ABB RAPID module: arm_code.mod

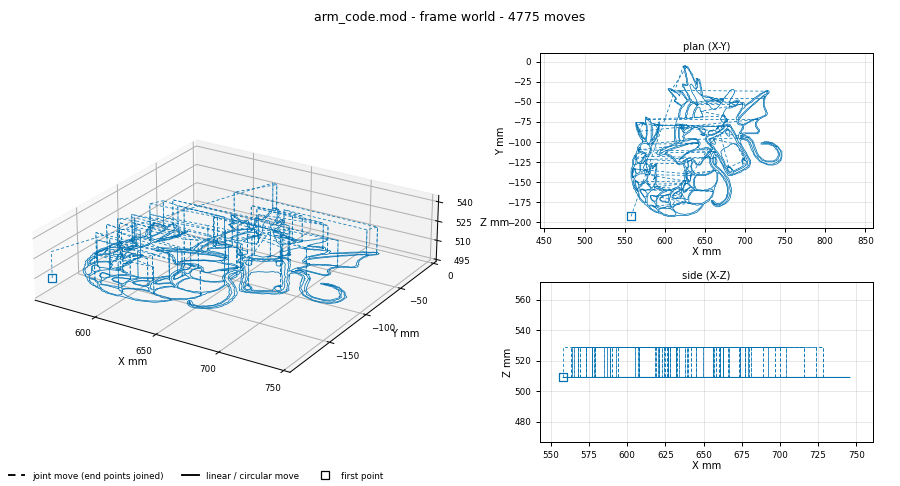
[picture p0: tool path of arm_code.mod in frame world, 4775 of 4775 moves have a stored position in this frame; points joined in program order, loops and branches not executed]
MODULE Module1
    !***********************************************************
    !
    ! Module:  Module1
    !
    ! Description:
    !   <Insert description here>
    !
    ! Author: ufabc
    !
    ! Version: 1.0
    !
    !***********************************************************


    !***********************************************************
    !
    ! Procedure main
    !
    !   This is the entry point of your program
    !
    !***********************************************************
    PROC main()
        !Add your code here
        CONST robtarget p0:=[[557.96,-192.62,509.20],[0.00299687,-0.165444,-0.986215,-0.000502744],[-1,0,0,0],[9E+09,9E+09,9E+09,9E+09,9E+09,9E+09]]
;
        MoveJ p0, v10, z1, tool0;
	MoveJ Offs(p0,0,0, 20), v10, z1, tool0;
	MoveJ Offs(p0,65.0,187.0, 20), v10, z1, tool0;
	MoveJ Offs(p0,65.0,187.0, 0), v10, z1, tool0;
	MoveL Offs(p0,66.0,184.0, 0), v10, z5, tool0;
	MoveL Offs(p0,66.0,184.0, 0), v10, z5, tool0;
	MoveL Offs(p0,66.0,184.0, 0), v10, z5, tool0;
	MoveL Offs(p0,67.0,181.0, 0), v10, z5, tool0;
	MoveL Offs(p0,67.0,179.0, 0), v10, z5, tool0;
	MoveL Offs(p0,68.0,176.0, 0), v10, z5, tool0;
	MoveL Offs(p0,68.0,174.0, 0), v10, z5, tool0;
	MoveL Offs(p0,69.0,172.0, 0), v10, z5, tool0;
	MoveL Offs(p0,69.0,169.0, 0), v10, z5, tool0;
	MoveL Offs(p0,69.0,167.0, 0), v10, z5, tool0;
	MoveL Offs(p0,70.0,165.0, 0), v10, z5, tool0;
	MoveL Offs(p0,70.0,164.0, 0), v10, z5, tool0;
	MoveL Offs(p0,70.0,163.0, 0), v10, z5, tool0;
	MoveL Offs(p0,68.0,164.0, 0), v10, z5, tool0;
	MoveL Offs(p0,66.0,165.0, 0), v10, z5, tool0;
	MoveL Offs(p0,65.0,165.0, 0), v10, z5, tool0;
	MoveL Offs(p0,65.0,165.0, 0), v10, z5, tool0;
	MoveL Offs(p0,64.0,165.0, 0), v10, z5, tool0;
	MoveL Offs(p0,64.0,165.0, 0), v10, z5, tool0;
	MoveL Offs(p0,64.0,165.0, 0), v10, z5, tool0;
	MoveL Offs(p0,64.0,165.0, 0), v10, z5, tool0;
	MoveL Offs(p0,64.0,162.0, 0), v10, z5, tool0;
	MoveL Offs(p0,65.0,161.0, 0), v10, z5, tool0;
	MoveL Offs(p0,65.0,161.0, 0), v10, z5, tool0;
	MoveL Offs(p0,66.0,160.0, 0), v10, z5, tool0;
	MoveL Offs(p0,68.0,156.0, 0), v10, z5, tool0;
	MoveL Offs(p0,69.0,155.0, 0), v10, z5, tool0;
	MoveL Offs(p0,70.0,153.0, 0), v10, z5, tool0;
	MoveL Offs(p0,70.0,151.0, 0), v10, z5, tool0;
	MoveL Offs(p0,71.0,150.0, 0), v10, z5, tool0;
	MoveL Offs(p0,72.0,149.0, 0), v10, z5, tool0;
	MoveL Offs(p0,72.0,147.0, 0), v10, z5, tool0;
	MoveL Offs(p0,73.0,147.0, 0), v10, z5, tool0;
	MoveL Offs(p0,73.0,146.0, 0), v10, z5, tool0;
	MoveL Offs(p0,71.0,145.0, 0), v10, z5, tool0;
	MoveL Offs(p0,69.0,147.0, 0), v10, z5, tool0;
	MoveL Offs(p0,69.0,148.0, 0), v10, z5, tool0;
	MoveL Offs(p0,68.0,148.0, 0), v10, z5, tool0;
	MoveL Offs(p0,67.0,151.0, 0), v10, z5, tool0;
	MoveL Offs(p0,66.0,152.0, 0), v10, z5, tool0;
	MoveL Offs(p0,66.0,152.0, 0), v10, z5, tool0;
	MoveL Offs(p0,65.0,153.0, 0), v10, z5, tool0;
	MoveL Offs(p0,65.0,154.0, 0), v10, z5, tool0;
	MoveL Offs(p0,64.0,154.0, 0), v10, z5, tool0;
	MoveL Offs(p0,64.0,155.0, 0), v10, z5, tool0;
	MoveL Offs(p0,62.0,157.0, 0), v10, z5, tool0;
	MoveL Offs(p0,61.0,157.0, 0), v10, z5, tool0;
	MoveL Offs(p0,61.0,157.0, 0), v10, z5, tool0;
	MoveL Offs(p0,61.0,157.0, 0), v10, z5, tool0;
	MoveL Offs(p0,61.0,157.0, 0), v10, z5, tool0;
	MoveL Offs(p0,60.0,157.0, 0), v10, z5, tool0;
	MoveL Offs(p0,60.0,155.0, 0), v10, z5, tool0;
	MoveL Offs(p0,57.0,155.0, 0), v10, z5, tool0;
	MoveL Offs(p0,56.0,155.0, 0), v10, z5, tool0;
	MoveL Offs(p0,55.0,156.0, 0), v10, z5, tool0;
	MoveL Offs(p0,53.0,157.0, 0), v10, z5, tool0;
	MoveL Offs(p0,52.0,158.0, 0), v10, z5, tool0;
	MoveL Offs(p0,51.0,158.0, 0), v10, z5, tool0;
	MoveL Offs(p0,50.0,159.0, 0), v10, z5, tool0;
	MoveL Offs(p0,49.0,159.0, 0), v10, z5, tool0;
	MoveL Offs(p0,49.0,159.0, 0), v10, z5, tool0;
	MoveL Offs(p0,46.0,159.0, 0), v10, z5, tool0;
	MoveL Offs(p0,46.0,159.0, 0), v10, z5, tool0;
	MoveL Offs(p0,46.0,159.0, 0), v10, z5, tool0;
	MoveL Offs(p0,47.0,157.0, 0), v10, z5, tool0;
	MoveL Offs(p0,48.0,156.0, 0), v10, z5, tool0;
	MoveL Offs(p0,49.0,155.0, 0), v10, z5, tool0;
	MoveL Offs(p0,50.0,153.0, 0), v10, z5, tool0;
	MoveL Offs(p0,52.0,151.0, 0), v10, z5, tool0;
	MoveL Offs(p0,57.0,146.0, 0), v10, z5, tool0;
	MoveL Offs(p0,55.0,146.0, 0), v10, z5, tool0;
	MoveL Offs(p0,54.0,144.0, 0), v10, z5, tool0;
	MoveL Offs(p0,54.0,143.0, 0), v10, z5, tool0;
	MoveL Offs(p0,55.0,143.0, 0), v10, z5, tool0;
	MoveL Offs(p0,57.0,141.0, 0), v10, z5, tool0;
	MoveL Offs(p0,58.0,141.0, 0), v10, z5, tool0;
	MoveL Offs(p0,58.0,140.0, 0), v10, z5, tool0;
	MoveL Offs(p0,59.0,140.0, 0), v10, z5, tool0;
	MoveL Offs(p0,59.0,140.0, 0), v10, z5, tool0;
	MoveL Offs(p0,63.0,137.0, 0), v10, z5, tool0;
	MoveL Offs(p0,61.0,134.0, 0), v10, z5, tool0;
	MoveL Offs(p0,60.0,132.0, 0), v10, z5, tool0;
	MoveL Offs(p0,60.0,130.0, 0), v10, z5, tool0;
	MoveL Offs(p0,60.0,129.0, 0), v10, z5, tool0;
	MoveL Offs(p0,59.0,128.0, 0), v10, z5, tool0;
	MoveL Offs(p0,59.0,127.0, 0), v10, z5, tool0;
	MoveL Offs(p0,59.0,126.0, 0), v10, z5, tool0;
	MoveL Offs(p0,59.0,125.0, 0), v10, z5, tool0;
	MoveL Offs(p0,59.0,124.0, 0), v10, z5, tool0;
	MoveL Offs(p0,58.0,122.0, 0), v10, z5, tool0;
	MoveL Offs(p0,58.0,122.0, 0), v10, z5, tool0;
	MoveL Offs(p0,58.0,122.0, 0), v10, z5, tool0;
	MoveL Offs(p0,58.0,122.0, 0), v10, z5, tool0;
	MoveL Offs(p0,56.0,117.0, 0), v10, z5, tool0;
	MoveL Offs(p0,56.0,116.0, 0), v10, z5, tool0;
	MoveL Offs(p0,56.0,116.0, 0), v10, z5, tool0;
	MoveL Offs(p0,56.0,115.0, 0), v10, z5, tool0;
	MoveL Offs(p0,55.0,114.0, 0), v10, z5, tool0;
	MoveL Offs(p0,55.0,114.0, 0), v10, z5, tool0;
	MoveL Offs(p0,54.0,111.0, 0), v10, z5, tool0;
	MoveL Offs(p0,54.0,111.0, 0), v10, z5, tool0;
	MoveL Offs(p0,54.0,110.0, 0), v10, z5, tool0;
	MoveL Offs(p0,54.0,109.0, 0), v10, z5, tool0;
	MoveL Offs(p0,54.0,108.0, 0), v10, z5, tool0;
	MoveL Offs(p0,54.0,107.0, 0), v10, z5, tool0;
	MoveL Offs(p0,54.0,106.0, 0), v10, z5, tool0;
	MoveL Offs(p0,54.0,104.0, 0), v10, z5, tool0;
	MoveL Offs(p0,54.0,101.0, 0), v10, z5, tool0;
	MoveL Offs(p0,54.0,100.0, 0), v10, z5, tool0;
	MoveL Offs(p0,54.0,99.0, 0), v10, z5, tool0;
	MoveL Offs(p0,54.0,97.0, 0), v10, z5, tool0;
	MoveL Offs(p0,54.0,96.0, 0), v10, z5, tool0;
	MoveL Offs(p0,54.0,95.0, 0), v10, z5, tool0;
	MoveL Offs(p0,54.0,94.0, 0), v10, z5, tool0;
	MoveL Offs(p0,55.0,93.0, 0), v10, z5, tool0;
	MoveL Offs(p0,55.0,92.0, 0), v10, z5, tool0;
	MoveL Offs(p0,53.0,90.0, 0), v10, z5, tool0;
	MoveL Offs(p0,52.0,90.0, 0), v10, z5, tool0;
	MoveL Offs(p0,50.0,89.0, 0), v10, z5, tool0;
	MoveL Offs(p0,49.0,88.0, 0), v10, z5, tool0;
	MoveL Offs(p0,46.0,87.0, 0), v10, z5, tool0;
	MoveL Offs(p0,44.0,86.0, 0), v10, z5, tool0;
	MoveL Offs(p0,41.0,86.0, 0), v10, z5, tool0;
	MoveL Offs(p0,40.0,85.0, 0), v10, z5, tool0;
	MoveL Offs(p0,38.0,84.0, 0), v10, z5, tool0;
	MoveL Offs(p0,36.0,83.0, 0), v10, z5, tool0;
	MoveL Offs(p0,35.0,83.0, 0), v10, z5, tool0;
	MoveL Offs(p0,34.0,82.0, 0), v10, z5, tool0;
	MoveL Offs(p0,34.0,82.0, 0), v10, z5, tool0;
	MoveL Offs(p0,33.0,81.0, 0), v10, z5, tool0;
	MoveL Offs(p0,32.0,79.0, 0), v10, z5, tool0;
	MoveL Offs(p0,32.0,78.0, 0), v10, z5, tool0;
	MoveL Offs(p0,32.0,78.0, 0), v10, z5, tool0;
	MoveL Offs(p0,32.0,78.0, 0), v10, z5, tool0;
	MoveL Offs(p0,33.0,77.0, 0), v10, z5, tool0;
	MoveL Offs(p0,33.0,77.0, 0), v10, z5, tool0;
	MoveL Offs(p0,36.0,76.0, 0), v10, z5, tool0;
	MoveL Offs(p0,36.0,76.0, 0), v10, z5, tool0;
	MoveL Offs(p0,36.0,76.0, 0), v10, z5, tool0;
	MoveL Offs(p0,37.0,76.0, 0), v10, z5, tool0;
	MoveL Offs(p0,37.0,76.0, 0), v10, z5, tool0;
	MoveL Offs(p0,40.0,77.0, 0), v10, z5, tool0;
	MoveL Offs(p0,41.0,77.0, 0), v10, z5, tool0;
	MoveL Offs(p0,42.0,77.0, 0), v10, z5, tool0;
	MoveL Offs(p0,44.0,77.0, 0), v10, z5, tool0;
	MoveL Offs(p0,45.0,76.0, 0), v10, z5, tool0;
	MoveL Offs(p0,47.0,76.0, 0), v10, z5, tool0;
	MoveL Offs(p0,48.0,75.0, 0), v10, z5, tool0;
	MoveL Offs(p0,49.0,74.0, 0), v10, z5, tool0;
	MoveL Offs(p0,51.0,73.0, 0), v10, z5, tool0;
	MoveL Offs(p0,52.0,72.0, 0), v10, z5, tool0;
	MoveL Offs(p0,53.0,71.0, 0), v10, z5, tool0;
	MoveL Offs(p0,53.0,71.0, 0), v10, z5, tool0;
	MoveL Offs(p0,54.0,70.0, 0), v10, z5, tool0;
	MoveL Offs(p0,55.0,69.0, 0), v10, z5, tool0;
	MoveL Offs(p0,55.0,68.0, 0), v10, z5, tool0;
	MoveL Offs(p0,56.0,68.0, 0), v10, z5, tool0;
	MoveL Offs(p0,58.0,65.0, 0), v10, z5, tool0;
	MoveL Offs(p0,58.0,65.0, 0), v10, z5, tool0;
	MoveL Offs(p0,59.0,65.0, 0), v10, z5, tool0;
	MoveL Offs(p0,60.0,64.0, 0), v10, z5, tool0;
	MoveL Offs(p0,60.0,64.0, 0), v10, z5, tool0;
	MoveL Offs(p0,61.0,65.0, 0), v10, z5, tool0;
	MoveL Offs(p0,62.0,65.0, 0), v10, z5, tool0;
	MoveL Offs(p0,63.0,65.0, 0), v10, z5, tool0;
	MoveL Offs(p0,64.0,66.0, 0), v10, z5, tool0;
	MoveL Offs(p0,65.0,64.0, 0), v10, z5, tool0;
	MoveL Offs(p0,66.0,62.0, 0), v10, z5, tool0;
	MoveL Offs(p0,66.0,62.0, 0), v10, z5, tool0;
	MoveL Offs(p0,66.0,61.0, 0), v10, z5, tool0;
	MoveL Offs(p0,66.0,61.0, 0), v10, z5, tool0;
	MoveL Offs(p0,67.0,61.0, 0), v10, z5, tool0;
	MoveL Offs(p0,67.0,59.0, 0), v10, z5, tool0;
	MoveL Offs(p0,67.0,58.0, 0), v10, z5, tool0;
	MoveL Offs(p0,67.0,58.0, 0), v10, z5, tool0;
	MoveL Offs(p0,66.0,56.0, 0), v10, z5, tool0;
	MoveL Offs(p0,66.0,55.0, 0), v10, z5, tool0;
	MoveL Offs(p0,66.0,54.0, 0), v10, z5, tool0;
	MoveL Offs(p0,66.0,53.0, 0), v10, z5, tool0;
	MoveL Offs(p0,66.0,52.0, 0), v10, z5, tool0;
	MoveL Offs(p0,66.0,51.0, 0), v10, z5, tool0;
	MoveL Offs(p0,66.0,50.0, 0), v10, z5, tool0;
	MoveL Offs(p0,66.0,50.0, 0), v10, z5, tool0;
	MoveL Offs(p0,67.0,47.0, 0), v10, z5, tool0;
	MoveL Offs(p0,66.0,45.0, 0), v10, z5, tool0;
	MoveL Offs(p0,64.0,43.0, 0), v10, z5, tool0;
	MoveL Offs(p0,63.0,42.0, 0), v10, z5, tool0;
	MoveL Offs(p0,63.0,41.0, 0), v10, z5, tool0;
	MoveL Offs(p0,62.0,40.0, 0), v10, z5, tool0;
	MoveL Offs(p0,62.0,40.0, 0), v10, z5, tool0;
	MoveL Offs(p0,62.0,39.0, 0), v10, z5, tool0;
	MoveL Offs(p0,62.0,39.0, 0), v10, z5, tool0;
	MoveL Offs(p0,58.0,37.0, 0), v10, z5, tool0;
	MoveL Offs(p0,57.0,36.0, 0), v10, z5, tool0;
	MoveL Offs(p0,56.0,36.0, 0), v10, z5, tool0;
	MoveL Offs(p0,55.0,36.0, 0), v10, z5, tool0;
	MoveL Offs(p0,54.0,35.0, 0), v10, z5, tool0;
	MoveL Offs(p0,54.0,35.0, 0), v10, z5, tool0;
	MoveL Offs(p0,53.0,34.0, 0), v10, z5, tool0;
	MoveL Offs(p0,53.0,34.0, 0), v10, z5, tool0;
	MoveL Offs(p0,50.0,33.0, 0), v10, z5, tool0;
	MoveL Offs(p0,50.0,33.0, 0), v10, z5, tool0;
	MoveL Offs(p0,49.0,33.0, 0), v10, z5, tool0;
	MoveL Offs(p0,49.0,33.0, 0), v10, z5, tool0;
	MoveL Offs(p0,47.0,33.0, 0), v10, z5, tool0;
	MoveL Offs(p0,46.0,33.0, 0), v10, z5, tool0;
	MoveL Offs(p0,46.0,33.0, 0), v10, z5, tool0;
	MoveL Offs(p0,45.0,33.0, 0), v10, z5, tool0;
	MoveL Offs(p0,45.0,33.0, 0), v10, z5, tool0;
	MoveL Offs(p0,45.0,33.0, 0), v10, z5, tool0;
	MoveL Offs(p0,42.0,33.0, 0), v10, z5, tool0;
	MoveL Offs(p0,42.0,33.0, 0), v10, z5, tool0;
	MoveL Offs(p0,42.0,33.0, 0), v10, z5, tool0;
	MoveL Offs(p0,42.0,33.0, 0), v10, z5, tool0;
	MoveL Offs(p0,41.0,33.0, 0), v10, z5, tool0;
	MoveL Offs(p0,39.0,35.0, 0), v10, z5, tool0;
	MoveL Offs(p0,38.0,35.0, 0), v10, z5, tool0;
	MoveL Offs(p0,37.0,35.0, 0), v10, z5, tool0;
	MoveL Offs(p0,37.0,35.0, 0), v10, z5, tool0;
	MoveL Offs(p0,36.0,36.0, 0), v10, z5, tool0;
	MoveL Offs(p0,35.0,36.0, 0), v10, z5, tool0;
	MoveL Offs(p0,33.0,37.0, 0), v10, z5, tool0;
	MoveL Offs(p0,33.0,37.0, 0), v10, z5, tool0;
	MoveL Offs(p0,33.0,38.0, 0), v10, z5, tool0;
	MoveL Offs(p0,31.0,40.0, 0), v10, z5, tool0;
	MoveL Offs(p0,31.0,40.0, 0), v10, z5, tool0;
	MoveL Offs(p0,31.0,42.0, 0), v10, z5, tool0;
	MoveL Offs(p0,31.0,43.0, 0), v10, z5, tool0;
	MoveL Offs(p0,31.0,44.0, 0), v10, z5, tool0;
	MoveL Offs(p0,32.0,46.0, 0), v10, z5, tool0;
	MoveL Offs(p0,32.0,47.0, 0), v10, z5, tool0;
	MoveL Offs(p0,32.0,48.0, 0), v10, z5, tool0;
	MoveL Offs(p0,32.0,49.0, 0), v10, z5, tool0;
	MoveL Offs(p0,32.0,49.0, 0), v10, z5, tool0;
	MoveL Offs(p0,32.0,50.0, 0), v10, z5, tool0;
	MoveL Offs(p0,32.0,50.0, 0), v10, z5, tool0;
	MoveL Offs(p0,32.0,51.0, 0), v10, z5, tool0;
	MoveL Offs(p0,31.0,51.0, 0), v10, z5, tool0;
	MoveL Offs(p0,31.0,53.0, 0), v10, z5, tool0;
	MoveL Offs(p0,31.0,55.0, 0), v10, z5, tool0;
	MoveL Offs(p0,31.0,56.0, 0), v10, z5, tool0;
	MoveL Offs(p0,31.0,57.0, 0), v10, z5, tool0;
	MoveL Offs(p0,31.0,58.0, 0), v10, z5, tool0;
	MoveL Offs(p0,32.0,58.0, 0), v10, z5, tool0;
	MoveL Offs(p0,32.0,59.0, 0), v10, z5, tool0;
	MoveL Offs(p0,32.0,60.0, 0), v10, z5, tool0;
	MoveL Offs(p0,32.0,62.0, 0), v10, z5, tool0;
	MoveL Offs(p0,32.0,63.0, 0), v10, z5, tool0;
	MoveL Offs(p0,32.0,63.0, 0), v10, z5, tool0;
	MoveL Offs(p0,32.0,64.0, 0), v10, z5, tool0;
	MoveL Offs(p0,32.0,64.0, 0), v10, z5, tool0;
	MoveL Offs(p0,32.0,65.0, 0), v10, z5, tool0;
	MoveL Offs(p0,32.0,65.0, 0), v10, z5, tool0;
	MoveL Offs(p0,32.0,65.0, 0), v10, z5, tool0;
	MoveL Offs(p0,32.0,65.0, 0), v10, z5, tool0;
	MoveL Offs(p0,29.0,65.0, 0), v10, z5, tool0;
	MoveL Offs(p0,29.0,65.0, 0), v10, z5, tool0;
	MoveL Offs(p0,29.0,64.0, 0), v10, z5, tool0;
	MoveL Offs(p0,28.0,63.0, 0), v10, z5, tool0;
	MoveL Offs(p0,27.0,61.0, 0), v10, z5, tool0;
	MoveL Offs(p0,26.0,63.0, 0), v10, z5, tool0;
	MoveL Offs(p0,25.0,65.0, 0), v10, z5, tool0;
	MoveL Offs(p0,25.0,65.0, 0), v10, z5, tool0;
	MoveL Offs(p0,25.0,65.0, 0), v10, z5, tool0;
	MoveL Offs(p0,25.0,65.0, 0), v10, z5, tool0;
	MoveL Offs(p0,23.0,63.0, 0), v10, z5, tool0;
	MoveL Offs(p0,23.0,63.0, 0), v10, z5, tool0;
	MoveL Offs(p0,23.0,60.0, 0), v10, z5, tool0;
	MoveL Offs(p0,23.0,59.0, 0), v10, z5, tool0;
	MoveL Offs(p0,23.0,58.0, 0), v10, z5, tool0;
	MoveL Offs(p0,23.0,58.0, 0), v10, z5, tool0;
	MoveL Offs(p0,23.0,57.0, 0), v10, z5, tool0;
	MoveL Offs(p0,23.0,57.0, 0), v10, z5, tool0;
	MoveL Offs(p0,23.0,56.0, 0), v10, z5, tool0;
	MoveL Offs(p0,23.0,56.0, 0), v10, z5, tool0;
	MoveL Offs(p0,23.0,56.0, 0), v10, z5, tool0;
	MoveL Offs(p0,20.0,55.0, 0), v10, z5, tool0;
	MoveL Offs(p0,20.0,56.0, 0), v10, z5, tool0;
	MoveL Offs(p0,20.0,58.0, 0), v10, z5, tool0;
	MoveL Offs(p0,20.0,59.0, 0), v10, z5, tool0;
	MoveL Offs(p0,20.0,60.0, 0), v10, z5, tool0;
	MoveL Offs(p0,20.0,60.0, 0), v10, z5, tool0;
	MoveL Offs(p0,20.0,60.0, 0), v10, z5, tool0;
	MoveL Offs(p0,20.0,61.0, 0), v10, z5, tool0;
	MoveL Offs(p0,19.0,61.0, 0), v10, z5, tool0;
	MoveL Offs(p0,19.0,63.0, 0), v10, z5, tool0;
	MoveL Offs(p0,19.0,64.0, 0), v10, z5, tool0;
	MoveL Offs(p0,19.0,64.0, 0), v10, z5, tool0;
	MoveL Offs(p0,19.0,65.0, 0), v10, z5, tool0;
	MoveL Offs(p0,19.0,66.0, 0), v10, z5, tool0;
	MoveL Offs(p0,19.0,66.0, 0), v10, z5, tool0;
	MoveL Offs(p0,19.0,67.0, 0), v10, z5, tool0;
	MoveL Offs(p0,20.0,69.0, 0), v10, z5, tool0;
	MoveL Offs(p0,20.0,69.0, 0), v10, z5, tool0;
	MoveL Offs(p0,20.0,70.0, 0), v10, z5, tool0;
	MoveL Offs(p0,20.0,70.0, 0), v10, z5, tool0;
	MoveL Offs(p0,20.0,71.0, 0), v10, z5, tool0;
	MoveL Offs(p0,20.0,71.0, 0), v10, z5, tool0;
	MoveL Offs(p0,21.0,73.0, 0), v10, z5, tool0;
	MoveL Offs(p0,21.0,74.0, 0), v10, z5, tool0;
	MoveL Offs(p0,21.0,74.0, 0), v10, z5, tool0;
	MoveL Offs(p0,21.0,74.0, 0), v10, z5, tool0;
	MoveL Offs(p0,22.0,75.0, 0), v10, z5, tool0;
	MoveL Offs(p0,22.0,75.0, 0), v10, z5, tool0;
	MoveL Offs(p0,23.0,77.0, 0), v10, z5, tool0;
	MoveL Offs(p0,24.0,78.0, 0), v10, z5, tool0;
	MoveL Offs(p0,24.0,79.0, 0), v10, z5, tool0;
	MoveL Offs(p0,24.0,80.0, 0), v10, z5, tool0;
	MoveL Offs(p0,25.0,81.0, 0), v10, z5, tool0;
	MoveL Offs(p0,25.0,82.0, 0), v10, z5, tool0;
	MoveL Offs(p0,25.0,83.0, 0), v10, z5, tool0;
	MoveL Offs(p0,25.0,85.0, 0), v10, z5, tool0;
	MoveL Offs(p0,25.0,87.0, 0), v10, z5, tool0;
	MoveL Offs(p0,25.0,87.0, 0), v10, z5, tool0;
	MoveL Offs(p0,25.0,88.0, 0), v10, z5, tool0;
	MoveL Offs(p0,25.0,88.0, 0), v10, z5, tool0;
	MoveL Offs(p0,25.0,88.0, 0), v10, z5, tool0;
	MoveL Offs(p0,26.0,88.0, 0), v10, z5, tool0;
	MoveL Offs(p0,26.0,89.0, 0), v10, z5, tool0;
	MoveL Offs(p0,26.0,89.0, 0), v10, z5, tool0;
	MoveL Offs(p0,28.0,91.0, 0), v10, z5, tool0;
	MoveL Offs(p0,28.0,92.0, 0), v10, z5, tool0;
	MoveL Offs(p0,29.0,93.0, 0), v10, z5, tool0;
	MoveL Offs(p0,30.0,94.0, 0), v10, z5, tool0;
	MoveL Offs(p0,30.0,95.0, 0), v10, z5, tool0;
	MoveL Offs(p0,31.0,96.0, 0), v10, z5, tool0;
	MoveL Offs(p0,31.0,97.0, 0), v10, z5, tool0;
	MoveL Offs(p0,32.0,97.0, 0), v10, z5, tool0;
	MoveL Offs(p0,33.0,101.0, 0), v10, z5, tool0;
	MoveL Offs(p0,34.0,103.0, 0), v10, z5, tool0;
	MoveL Offs(p0,34.0,105.0, 0), v10, z5, tool0;
	MoveL Offs(p0,35.0,106.0, 0), v10, z5, tool0;
	MoveL Offs(p0,35.0,108.0, 0), v10, z5, tool0;
	MoveL Offs(p0,35.0,110.0, 0), v10, z5, tool0;
	MoveL Offs(p0,35.0,112.0, 0), v10, z5, tool0;
	MoveL Offs(p0,36.0,114.0, 0), v10, z5, tool0;
	MoveL Offs(p0,36.0,115.0, 0), v10, z5, tool0;
	MoveL Offs(p0,35.0,117.0, 0), v10, z5, tool0;
	MoveL Offs(p0,35.0,118.0, 0), v10, z5, tool0;
	MoveL Offs(p0,35.0,118.0, 0), v10, z5, tool0;
	MoveL Offs(p0,35.0,118.0, 0), v10, z5, tool0;
	MoveL Offs(p0,35.0,118.0, 0), v10, z5, tool0;
	MoveL Offs(p0,35.0,118.0, 0), v10, z5, tool0;
	MoveL Offs(p0,34.0,116.0, 0), v10, z5, tool0;
	MoveL Offs(p0,33.0,114.0, 0), v10, z5, tool0;
	MoveL Offs(p0,33.0,114.0, 0), v10, z5, tool0;
	MoveL Offs(p0,33.0,113.0, 0), v10, z5, tool0;
	MoveL Offs(p0,33.0,113.0, 0), v10, z5, tool0;
	MoveL Offs(p0,33.0,114.0, 0), v10, z5, tool0;
	MoveL Offs(p0,28.0,116.0, 0), v10, z5, tool0;
	MoveL Offs(p0,27.0,115.0, 0), v10, z5, tool0;
	MoveL Offs(p0,25.0,117.0, 0), v10, z5, tool0;
	MoveL Offs(p0,24.0,119.0, 0), v10, z5, tool0;
	MoveL Offs(p0,24.0,120.0, 0), v10, z5, tool0;
	MoveL Offs(p0,24.0,120.0, 0), v10, z5, tool0;
	MoveL Offs(p0,23.0,121.0, 0), v10, z5, tool0;
	MoveL Offs(p0,23.0,121.0, 0), v10, z5, tool0;
	MoveL Offs(p0,23.0,122.0, 0), v10, z5, tool0;
	MoveL Offs(p0,22.0,122.0, 0), v10, z5, tool0;
	MoveL Offs(p0,22.0,122.0, 0), v10, z5, tool0;
	MoveL Offs(p0,18.0,124.0, 0), v10, z5, tool0;
	MoveL Offs(p0,18.0,124.0, 0), v10, z5, tool0;
	MoveL Offs(p0,18.0,124.0, 0), v10, z5, tool0;
	MoveL Offs(p0,18.0,124.0, 0), v10, z5, tool0;
	MoveL Offs(p0,18.0,124.0, 0), v10, z5, tool0;
	MoveL Offs(p0,18.0,122.0, 0), v10, z5, tool0;
	MoveL Offs(p0,18.0,117.0, 0), v10, z5, tool0;
	MoveL Offs(p0,17.0,116.0, 0), v10, z5, tool0;
	MoveL Offs(p0,17.0,116.0, 0), v10, z5, tool0;
	MoveL Offs(p0,17.0,116.0, 0), v10, z5, tool0;
	MoveL Offs(p0,14.0,117.0, 0), v10, z5, tool0;
	MoveL Offs(p0,14.0,116.0, 0), v10, z5, tool0;
	MoveL Offs(p0,13.0,117.0, 0), v10, z5, tool0;
	MoveL Offs(p0,6.0,117.0, 0), v10, z5, tool0;
	MoveL Offs(p0,6.0,116.0, 0), v10, z5, tool0;
	MoveL Offs(p0,6.0,112.0, 0), v10, z5, tool0;
	MoveL Offs(p0,7.0,110.0, 0), v10, z5, tool0;
	MoveL Offs(p0,7.0,108.0, 0), v10, z5, tool0;
	MoveL Offs(p0,8.0,106.0, 0), v10, z5, tool0;
	MoveL Offs(p0,9.0,104.0, 0), v10, z5, tool0;
	MoveL Offs(p0,9.0,102.0, 0), v10, z5, tool0;
	MoveL Offs(p0,10.0,101.0, 0), v10, z5, tool0;
	MoveL Offs(p0,11.0,99.0, 0), v10, z5, tool0;
	MoveL Offs(p0,12.0,97.0, 0), v10, z5, tool0;
	MoveL Offs(p0,14.0,95.0, 0), v10, z5, tool0;
	MoveL Offs(p0,14.0,94.0, 0), v10, z5, tool0;
	MoveL Offs(p0,14.0,93.0, 0), v10, z5, tool0;
	MoveL Offs(p0,14.0,93.0, 0), v10, z5, tool0;
	MoveL Offs(p0,15.0,93.0, 0), v10, z5, tool0;
	MoveL Offs(p0,14.0,92.0, 0), v10, z5, tool0;
	MoveL Offs(p0,14.0,92.0, 0), v10, z5, tool0;
	MoveL Offs(p0,14.0,92.0, 0), v10, z5, tool0;
	MoveL Offs(p0,14.0,92.0, 0), v10, z5, tool0;
	MoveL Offs(p0,11.0,90.0, 0), v10, z5, tool0;
	MoveL Offs(p0,10.0,89.0, 0), v10, z5, tool0;
	MoveL Offs(p0,10.0,88.0, 0), v10, z5, tool0;
	MoveL Offs(p0,9.0,87.0, 0), v10, z5, tool0;
	MoveL Offs(p0,8.0,86.0, 0), v10, z5, tool0;
	MoveL Offs(p0,8.0,84.0, 0), v10, z5, tool0;
	MoveL Offs(p0,8.0,83.0, 0), v10, z5, tool0;
	MoveL Offs(p0,7.0,81.0, 0), v10, z5, tool0;
	MoveL Offs(p0,7.0,79.0, 0), v10, z5, tool0;
	MoveL Offs(p0,7.0,79.0, 0), v10, z5, tool0;
	MoveL Offs(p0,7.0,79.0, 0), v10, z5, tool0;
	MoveL Offs(p0,7.0,79.0, 0), v10, z5, tool0;
	MoveL Offs(p0,6.0,78.0, 0), v10, z5, tool0;
	MoveL Offs(p0,6.0,78.0, 0), v10, z5, tool0;
	MoveL Offs(p0,5.0,76.0, 0), v10, z5, tool0;
	MoveL Offs(p0,4.0,76.0, 0), v10, z5, tool0;
	MoveL Offs(p0,4.0,75.0, 0), v10, z5, tool0;
	MoveL Offs(p0,4.0,75.0, 0), v10, z5, tool0;
	MoveL Offs(p0,3.0,72.0, 0), v10, z5, tool0;
	MoveL Offs(p0,3.0,72.0, 0), v10, z5, tool0;
	MoveL Offs(p0,2.0,71.0, 0), v10, z5, tool0;
	MoveL Offs(p0,2.0,71.0, 0), v10, z5, tool0;
	MoveL Offs(p0,2.0,70.0, 0), v10, z5, tool0;
	MoveL Offs(p0,2.0,69.0, 0), v10, z5, tool0;
	MoveL Offs(p0,2.0,68.0, 0), v10, z5, tool0;
	MoveL Offs(p0,2.0,67.0, 0), v10, z5, tool0;
	MoveL Offs(p0,2.0,64.0, 0), v10, z5, tool0;
	MoveL Offs(p0,2.0,64.0, 0), v10, z5, tool0;
	MoveL Offs(p0,2.0,63.0, 0), v10, z5, tool0;
	MoveL Offs(p0,2.0,63.0, 0), v10, z5, tool0;
	MoveL Offs(p0,2.0,62.0, 0), v10, z5, tool0;
	MoveL Offs(p0,2.0,62.0, 0), v10, z5, tool0;
	MoveL Offs(p0,1.0,61.0, 0), v10, z5, tool0;
	MoveL Offs(p0,1.0,61.0, 0), v10, z5, tool0;
	MoveL Offs(p0,0.0,58.0, 0), v10, z5, tool0;
	MoveL Offs(p0,0.0,57.0, 0), v10, z5, tool0;
	MoveL Offs(p0,0.0,56.0, 0), v10, z5, tool0;
	MoveL Offs(p0,0.0,54.0, 0), v10, z5, tool0;
	MoveL Offs(p0,0.0,52.0, 0), v10, z5, tool0;
	MoveL Offs(p0,0.0,51.0, 0), v10, z5, tool0;
	MoveL Offs(p0,0.0,49.0, 0), v10, z5, tool0;
	MoveL Offs(p0,0.0,48.0, 0), v10, z5, tool0;
	MoveL Offs(p0,1.0,47.0, 0), v10, z5, tool0;
	MoveL Offs(p0,1.0,44.0, 0), v10, z5, tool0;
	MoveL Offs(p0,1.0,44.0, 0), v10, z5, tool0;
	MoveL Offs(p0,2.0,43.0, 0), v10, z5, tool0;
	MoveL Offs(p0,2.0,43.0, 0), v10, z5, tool0;
	MoveL Offs(p0,2.0,43.0, 0), v10, z5, tool0;
	MoveL Offs(p0,2.0,42.0, 0), v10, z5, tool0;
	MoveL Offs(p0,2.0,40.0, 0), v10, z5, tool0;
	MoveL Offs(p0,2.0,39.0, 0), v10, z5, tool0;
	MoveL Offs(p0,3.0,38.0, 0), v10, z5, tool0;
	MoveL Offs(p0,3.0,36.0, 0), v10, z5, tool0;
	MoveL Offs(p0,3.0,35.0, 0), v10, z5, tool0;
	MoveL Offs(p0,4.0,34.0, 0), v10, z5, tool0;
	MoveL Offs(p0,4.0,34.0, 0), v10, z5, tool0;
	MoveL Offs(p0,5.0,33.0, 0), v10, z5, tool0;
	MoveL Offs(p0,6.0,30.0, 0), v10, z5, tool0;
	MoveL Offs(p0,6.0,30.0, 0), v10, z5, tool0;
	MoveL Offs(p0,7.0,30.0, 0), v10, z5, tool0;
	MoveL Offs(p0,7.0,29.0, 0), v10, z5, tool0;
	MoveL Offs(p0,8.0,27.0, 0), v10, z5, tool0;
	MoveL Offs(p0,8.0,27.0, 0), v10, z5, tool0;
	MoveL Offs(p0,8.0,27.0, 0), v10, z5, tool0;
	MoveL Offs(p0,8.0,27.0, 0), v10, z5, tool0;
	MoveL Offs(p0,9.0,25.0, 0), v10, z5, tool0;
	MoveL Offs(p0,9.0,24.0, 0), v10, z5, tool0;
	MoveL Offs(p0,10.0,24.0, 0), v10, z5, tool0;
	MoveL Offs(p0,11.0,21.0, 0), v10, z5, tool0;
	MoveL Offs(p0,12.0,20.0, 0), v10, z5, tool0;
	MoveL Offs(p0,13.0,19.0, 0), v10, z5, tool0;
	MoveL Offs(p0,14.0,18.0, 0), v10, z5, tool0;
	MoveL Offs(p0,15.0,17.0, 0), v10, z5, tool0;
	MoveL Offs(p0,16.0,17.0, 0), v10, z5, tool0;
	MoveL Offs(p0,17.0,16.0, 0), v10, z5, tool0;
	MoveL Offs(p0,17.0,15.0, 0), v10, z5, tool0;
	MoveL Offs(p0,19.0,14.0, 0), v10, z5, tool0;
	MoveL Offs(p0,20.0,14.0, 0), v10, z5, tool0;
	MoveL Offs(p0,20.0,14.0, 0), v10, z5, tool0;
	MoveL Offs(p0,20.0,13.0, 0), v10, z5, tool0;
	MoveL Offs(p0,22.0,11.0, 0), v10, z5, tool0;
	MoveL Offs(p0,23.0,10.0, 0), v10, z5, tool0;
	MoveL Offs(p0,24.0,9.0, 0), v10, z5, tool0;
	MoveL Offs(p0,26.0,8.0, 0), v10, z5, tool0;
	MoveL Offs(p0,27.0,7.0, 0), v10, z5, tool0;
	MoveL Offs(p0,29.0,6.0, 0), v10, z5, tool0;
	MoveL Offs(p0,31.0,5.0, 0), v10, z5, tool0;
	MoveL Offs(p0,33.0,5.0, 0), v10, z5, tool0;
	MoveL Offs(p0,34.0,4.0, 0), v10, z5, tool0;
	MoveL Offs(p0,37.0,4.0, 0), v10, z5, tool0;
	MoveL Offs(p0,37.0,3.0, 0), v10, z5, tool0;
	MoveL Offs(p0,38.0,3.0, 0), v10, z5, tool0;
	MoveL Offs(p0,38.0,3.0, 0), v10, z5, tool0;
	MoveL Offs(p0,39.0,3.0, 0), v10, z5, tool0;
	MoveL Offs(p0,39.0,3.0, 0), v10, z5, tool0;
	MoveL Offs(p0,41.0,1.0, 0), v10, z5, tool0;
	MoveL Offs(p0,43.0,1.0, 0), v10, z5, tool0;
	MoveL Offs(p0,44.0,1.0, 0), v10, z5, tool0;
	MoveL Offs(p0,45.0,0.0, 0), v10, z5, tool0;
	MoveL Offs(p0,46.0,0.0, 0), v10, z5, tool0;
	MoveL Offs(p0,47.0,0.0, 0), v10, z5, tool0;
	MoveL Offs(p0,49.0,0.0, 0), v10, z5, tool0;
	MoveL Offs(p0,50.0,0.0, 0), v10, z5, tool0;
	MoveL Offs(p0,52.0,0.0, 0), v10, z5, tool0;
	MoveL Offs(p0,54.0,0.0, 0), v10, z5, tool0;
	MoveL Offs(p0,55.0,0.0, 0), v10, z5, tool0;
	MoveL Offs(p0,55.0,0.0, 0), v10, z5, tool0;
	MoveL Offs(p0,56.0,1.0, 0), v10, z5, tool0;
	MoveL Offs(p0,57.0,1.0, 0), v10, z5, tool0;
	MoveL Offs(p0,57.0,1.0, 0), v10, z5, tool0;
	MoveL Offs(p0,58.0,1.0, 0), v10, z5, tool0;
	MoveL Offs(p0,58.0,1.0, 0), v10, z5, tool0;
	MoveL Offs(p0,60.0,1.0, 0), v10, z5, tool0;
	MoveL Offs(p0,61.0,1.0, 0), v10, z5, tool0;
	MoveL Offs(p0,61.0,1.0, 0), v10, z5, tool0;
	MoveL Offs(p0,62.0,1.0, 0), v10, z5, tool0;
	MoveL Offs(p0,62.0,1.0, 0), v10, z5, tool0;
	MoveL Offs(p0,63.0,1.0, 0), v10, z5, tool0;
	MoveL Offs(p0,66.0,1.0, 0), v10, z5, tool0;
	MoveL Offs(p0,70.0,1.0, 0), v10, z5, tool0;
	MoveL Offs(p0,73.0,2.0, 0), v10, z5, tool0;
	MoveL Offs(p0,76.0,3.0, 0), v10, z5, tool0;
	MoveL Offs(p0,79.0,4.0, 0), v10, z5, tool0;
	MoveL Offs(p0,82.0,5.0, 0), v10, z5, tool0;
	MoveL Offs(p0,84.0,7.0, 0), v10, z5, tool0;
	MoveL Offs(p0,86.0,9.0, 0), v10, z5, tool0;
	MoveL Offs(p0,88.0,11.0, 0), v10, z5, tool0;
	MoveL Offs(p0,90.0,14.0, 0), v10, z5, tool0;
	MoveL Offs(p0,91.0,16.0, 0), v10, z5, tool0;
	MoveL Offs(p0,92.0,16.0, 0), v10, z5, tool0;
	MoveL Offs(p0,92.0,16.0, 0), v10, z5, tool0;
	MoveL Offs(p0,93.0,17.0, 0), v10, z5, tool0;
	MoveL Offs(p0,93.0,17.0, 0), v10, z5, tool0;
	MoveL Offs(p0,97.0,19.0, 0), v10, z5, tool0;
	MoveL Offs(p0,98.0,21.0, 0), v10, z5, tool0;
	MoveL Offs(p0,99.0,23.0, 0), v10, z5, tool0;
	MoveL Offs(p0,101.0,24.0, 0), v10, z5, tool0;
	MoveL Offs(p0,102.0,26.0, 0), v10, z5, tool0;
	MoveL Offs(p0,102.0,28.0, 0), v10, z5, tool0;
	MoveL Offs(p0,103.0,30.0, 0), v10, z5, tool0;
	MoveL Offs(p0,103.0,32.0, 0), v10, z5, tool0;
	MoveL Offs(p0,104.0,34.0, 0), v10, z5, tool0;
	MoveL Offs(p0,104.0,36.0, 0), v10, z5, tool0;
	MoveL Offs(p0,104.0,37.0, 0), v10, z5, tool0;
	MoveL Offs(p0,104.0,37.0, 0), v10, z5, tool0;
	MoveL Offs(p0,105.0,37.0, 0), v10, z5, tool0;
	MoveL Offs(p0,105.0,38.0, 0), v10, z5, tool0;
	MoveL Offs(p0,106.0,40.0, 0), v10, z5, tool0;
	MoveL Offs(p0,107.0,42.0, 0), v10, z5, tool0;
	MoveL Offs(p0,107.0,43.0, 0), v10, z5, tool0;
	MoveL Offs(p0,108.0,45.0, 0), v10, z5, tool0;
	MoveL Offs(p0,108.0,47.0, 0), v10, z5, tool0;
	MoveL Offs(p0,108.0,48.0, 0), v10, z5, tool0;
	MoveL Offs(p0,108.0,50.0, 0), v10, z5, tool0;
	MoveL Offs(p0,108.0,51.0, 0), v10, z5, tool0;
	MoveL Offs(p0,108.0,53.0, 0), v10, z5, tool0;
	MoveL Offs(p0,108.0,55.0, 0), v10, z5, tool0;
	MoveL Offs(p0,108.0,55.0, 0), v10, z5, tool0;
	MoveL Offs(p0,108.0,55.0, 0), v10, z5, tool0;
	MoveL Offs(p0,108.0,55.0, 0), v10, z5, tool0;
	MoveL Offs(p0,110.0,53.0, 0), v10, z5, tool0;
	MoveL Offs(p0,110.0,53.0, 0), v10, z5, tool0;
	MoveL Offs(p0,111.0,53.0, 0), v10, z5, tool0;
	MoveL Offs(p0,113.0,50.0, 0), v10, z5, tool0;
	MoveL Offs(p0,114.0,49.0, 0), v10, z5, tool0;
	MoveL Offs(p0,115.0,48.0, 0), v10, z5, tool0;
	MoveL Offs(p0,115.0,47.0, 0), v10, z5, tool0;
	MoveL Offs(p0,116.0,45.0, 0), v10, z5, tool0;
	MoveL Offs(p0,117.0,44.0, 0), v10, z5, tool0;
	MoveL Offs(p0,118.0,43.0, 0), v10, z5, tool0;
	MoveL Offs(p0,118.0,42.0, 0), v10, z5, tool0;
	MoveL Offs(p0,119.0,40.0, 0), v10, z5, tool0;
	MoveL Offs(p0,119.0,38.0, 0), v10, z5, tool0;
	MoveL Offs(p0,120.0,37.0, 0), v10, z5, tool0;
	MoveL Offs(p0,120.0,37.0, 0), v10, z5, tool0;
	MoveL Offs(p0,120.0,36.0, 0), v10, z5, tool0;
	MoveL Offs(p0,120.0,35.0, 0), v10, z5, tool0;
	MoveL Offs(p0,120.0,34.0, 0), v10, z5, tool0;
	MoveL Offs(p0,120.0,33.0, 0), v10, z5, tool0;
	MoveL Offs(p0,120.0,32.0, 0), v10, z5, tool0;
	MoveL Offs(p0,120.0,30.0, 0), v10, z5, tool0;
	MoveL Offs(p0,120.0,29.0, 0), v10, z5, tool0;
	MoveL Offs(p0,120.0,29.0, 0), v10, z5, tool0;
	MoveL Offs(p0,120.0,28.0, 0), v10, z5, tool0;
	MoveL Offs(p0,120.0,27.0, 0), v10, z5, tool0;
	MoveL Offs(p0,119.0,27.0, 0), v10, z5, tool0;
	MoveL Offs(p0,119.0,26.0, 0), v10, z5, tool0;
	MoveL Offs(p0,119.0,26.0, 0), v10, z5, tool0;
	MoveL Offs(p0,119.0,25.0, 0), v10, z5, tool0;
	MoveL Offs(p0,118.0,22.0, 0), v10, z5, tool0;
	MoveL Offs(p0,117.0,21.0, 0), v10, z5, tool0;
	MoveL Offs(p0,117.0,21.0, 0), v10, z5, tool0;
	MoveL Offs(p0,116.0,20.0, 0), v10, z5, tool0;
	MoveL Offs(p0,115.0,19.0, 0), v10, z5, tool0;
	MoveL Offs(p0,115.0,19.0, 0), v10, z5, tool0;
	MoveL Offs(p0,114.0,18.0, 0), v10, z5, tool0;
	MoveL Offs(p0,113.0,18.0, 0), v10, z5, tool0;
	MoveL Offs(p0,111.0,16.0, 0), v10, z5, tool0;
	MoveL Offs(p0,109.0,16.0, 0), v10, z5, tool0;
	MoveL Offs(p0,108.0,16.0, 0), v10, z5, tool0;
	MoveL Offs(p0,107.0,16.0, 0), v10, z5, tool0;
	MoveL Offs(p0,106.0,16.0, 0), v10, z5, tool0;
	MoveL Offs(p0,105.0,17.0, 0), v10, z5, tool0;
	MoveL Offs(p0,104.0,18.0, 0), v10, z5, tool0;
	MoveL Offs(p0,103.0,19.0, 0), v10, z5, tool0;
	MoveL Offs(p0,102.0,20.0, 0), v10, z5, tool0;
	MoveL Offs(p0,100.0,20.0, 0), v10, z5, tool0;
	MoveL Offs(p0,100.0,19.0, 0), v10, z5, tool0;
	MoveL Offs(p0,100.0,18.0, 0), v10, z5, tool0;
	MoveL Offs(p0,100.0,18.0, 0), v10, z5, tool0;
	MoveL Offs(p0,101.0,17.0, 0), v10, z5, tool0;
	MoveL Offs(p0,101.0,16.0, 0), v10, z5, tool0;
	MoveL Offs(p0,103.0,14.0, 0), v10, z5, tool0;
	MoveL Offs(p0,104.0,13.0, 0), v10, z5, tool0;
	MoveL Offs(p0,105.0,13.0, 0), v10, z5, tool0;
	MoveL Offs(p0,106.0,12.0, 0), v10, z5, tool0;
	MoveL Offs(p0,107.0,12.0, 0), v10, z5, tool0;
	MoveL Offs(p0,108.0,12.0, 0), v10, z5, tool0;
	MoveL Offs(p0,109.0,12.0, 0), v10, z5, tool0;
	MoveL Offs(p0,110.0,12.0, 0), v10, z5, tool0;
	MoveL Offs(p0,112.0,13.0, 0), v10, z5, tool0;
	MoveL Offs(p0,114.0,14.0, 0), v10, z5, tool0;
	MoveL Offs(p0,116.0,15.0, 0), v10, z5, tool0;
	MoveL Offs(p0,118.0,16.0, 0), v10, z5, tool0;
	MoveL Offs(p0,119.0,17.0, 0), v10, z5, tool0;
	MoveL Offs(p0,121.0,19.0, 0), v10, z5, tool0;
	MoveL Offs(p0,122.0,20.0, 0), v10, z5, tool0;
	MoveL Offs(p0,123.0,22.0, 0), v10, z5, tool0;
	MoveL Offs(p0,124.0,24.0, 0), v10, z5, tool0;
	MoveL Offs(p0,124.0,26.0, 0), v10, z5, tool0;
	MoveL Offs(p0,125.0,29.0, 0), v10, z5, tool0;
	MoveL Offs(p0,125.0,31.0, 0), v10, z5, tool0;
	MoveL Offs(p0,125.0,32.0, 0), v10, z5, tool0;
	MoveL Offs(p0,125.0,34.0, 0), v10, z5, tool0;
	MoveL Offs(p0,125.0,36.0, 0), v10, z5, tool0;
	MoveL Offs(p0,124.0,37.0, 0), v10, z5, tool0;
	MoveL Offs(p0,124.0,39.0, 0), v10, z5, tool0;
	MoveL Offs(p0,124.0,40.0, 0), v10, z5, tool0;
	MoveL Offs(p0,123.0,42.0, 0), v10, z5, tool0;
	MoveL Offs(p0,123.0,44.0, 0), v10, z5, tool0;
	MoveL Offs(p0,122.0,46.0, 0), v10, z5, tool0;
	MoveL Offs(p0,121.0,48.0, 0), v10, z5, tool0;
	MoveL Offs(p0,119.0,50.0, 0), v10, z5, tool0;
	MoveL Offs(p0,118.0,51.0, 0), v10, z5, tool0;
	MoveL Offs(p0,117.0,53.0, 0), v10, z5, tool0;
	MoveL Offs(p0,115.0,55.0, 0), v10, z5, tool0;
	MoveL Offs(p0,113.0,57.0, 0), v10, z5, tool0;
	MoveL Offs(p0,112.0,58.0, 0), v10, z5, tool0;
	MoveL Offs(p0,110.0,60.0, 0), v10, z5, tool0;
	MoveL Offs(p0,106.0,63.0, 0), v10, z5, tool0;
	MoveL Offs(p0,106.0,65.0, 0), v10, z5, tool0;
	MoveL Offs(p0,107.0,68.0, 0), v10, z5, tool0;
	MoveL Offs(p0,107.0,69.0, 0), v10, z5, tool0;
	MoveL Offs(p0,107.0,70.0, 0), v10, z5, tool0;
	MoveL Offs(p0,107.0,70.0, 0), v10, z5, tool0;
	MoveL Offs(p0,106.0,71.0, 0), v10, z5, tool0;
	MoveL Offs(p0,106.0,72.0, 0), v10, z5, tool0;
	MoveL Offs(p0,106.0,73.0, 0), v10, z5, tool0;
	MoveL Offs(p0,106.0,74.0, 0), v10, z5, tool0;
	MoveL Offs(p0,105.0,77.0, 0), v10, z5, tool0;
	MoveL Offs(p0,105.0,77.0, 0), v10, z5, tool0;
	MoveL Offs(p0,106.0,77.0, 0), v10, z5, tool0;
	MoveL Offs(p0,106.0,77.0, 0), v10, z5, tool0;
	MoveL Offs(p0,106.0,77.0, 0), v10, z5, tool0;
	MoveL Offs(p0,106.0,77.0, 0), v10, z5, tool0;
	MoveL Offs(p0,108.0,74.0, 0), v10, z5, tool0;
	MoveL Offs(p0,109.0,73.0, 0), v10, z5, tool0;
	MoveL Offs(p0,110.0,71.0, 0), v10, z5, tool0;
	MoveL Offs(p0,111.0,69.0, 0), v10, z5, tool0;
	MoveL Offs(p0,112.0,67.0, 0), v10, z5, tool0;
	MoveL Offs(p0,114.0,64.0, 0), v10, z5, tool0;
	MoveL Offs(p0,115.0,61.0, 0), v10, z5, tool0;
	MoveL Offs(p0,116.0,59.0, 0), v10, z5, tool0;
	MoveL Offs(p0,117.0,57.0, 0), v10, z5, tool0;
	MoveL Offs(p0,118.0,55.0, 0), v10, z5, tool0;
	MoveL Offs(p0,119.0,54.0, 0), v10, z5, tool0;
	MoveL Offs(p0,120.0,53.0, 0), v10, z5, tool0;
	MoveL Offs(p0,120.0,52.0, 0), v10, z5, tool0;
	MoveL Offs(p0,121.0,51.0, 0), v10, z5, tool0;
	MoveL Offs(p0,122.0,51.0, 0), v10, z5, tool0;
	MoveL Offs(p0,122.0,51.0, 0), v10, z5, tool0;
	MoveL Offs(p0,123.0,51.0, 0), v10, z5, tool0;
	MoveL Offs(p0,125.0,51.0, 0), v10, z5, tool0;
	MoveL Offs(p0,126.0,51.0, 0), v10, z5, tool0;
	MoveL Offs(p0,128.0,52.0, 0), v10, z5, tool0;
	MoveL Offs(p0,129.0,52.0, 0), v10, z5, tool0;
	MoveL Offs(p0,131.0,53.0, 0), v10, z5, tool0;
	MoveL Offs(p0,133.0,54.0, 0), v10, z5, tool0;
	MoveL Offs(p0,134.0,54.0, 0), v10, z5, tool0;
	MoveL Offs(p0,137.0,55.0, 0), v10, z5, tool0;
	MoveL Offs(p0,139.0,57.0, 0), v10, z5, tool0;
	MoveL Offs(p0,141.0,58.0, 0), v10, z5, tool0;
	MoveL Offs(p0,142.0,58.0, 0), v10, z5, tool0;
	MoveL Offs(p0,144.0,59.0, 0), v10, z5, tool0;
	MoveL Offs(p0,145.0,60.0, 0), v10, z5, tool0;
	MoveL Offs(p0,146.0,61.0, 0), v10, z5, tool0;
	MoveL Offs(p0,147.0,61.0, 0), v10, z5, tool0;
	MoveL Offs(p0,147.0,62.0, 0), v10, z5, tool0;
	MoveL Offs(p0,148.0,63.0, 0), v10, z5, tool0;
	MoveL Offs(p0,148.0,64.0, 0), v10, z5, tool0;
	MoveL Offs(p0,149.0,66.0, 0), v10, z5, tool0;
	MoveL Offs(p0,149.0,67.0, 0), v10, z5, tool0;
	MoveL Offs(p0,149.0,68.0, 0), v10, z5, tool0;
	MoveL Offs(p0,149.0,70.0, 0), v10, z5, tool0;
	MoveL Offs(p0,148.0,71.0, 0), v10, z5, tool0;
	MoveL Offs(p0,147.0,73.0, 0), v10, z5, tool0;
	MoveL Offs(p0,145.0,76.0, 0), v10, z5, tool0;
	MoveL Offs(p0,144.0,79.0, 0), v10, z5, tool0;
	MoveL Offs(p0,141.0,83.0, 0), v10, z5, tool0;
	MoveL Offs(p0,140.0,85.0, 0), v10, z5, tool0;
	MoveL Offs(p0,139.0,87.0, 0), v10, z5, tool0;
	MoveL Offs(p0,138.0,88.0, 0), v10, z5, tool0;
	MoveL Offs(p0,138.0,89.0, 0), v10, z5, tool0;
	MoveL Offs(p0,137.0,90.0, 0), v10, z5, tool0;
	MoveL Offs(p0,137.0,91.0, 0), v10, z5, tool0;
	MoveL Offs(p0,136.0,91.0, 0), v10, z5, tool0;
	MoveL Offs(p0,136.0,92.0, 0), v10, z5, tool0;
	MoveL Offs(p0,136.0,92.0, 0), v10, z5, tool0;
	MoveL Offs(p0,136.0,94.0, 0), v10, z5, tool0;
	MoveL Offs(p0,138.0,96.0, 0), v10, z5, tool0;
	MoveL Offs(p0,139.0,96.0, 0), v10, z5, tool0;
	MoveL Offs(p0,140.0,96.0, 0), v10, z5, tool0;
	MoveL Offs(p0,141.0,96.0, 0), v10, z5, tool0;
	MoveL Offs(p0,142.0,95.0, 0), v10, z5, tool0;
	MoveL Offs(p0,143.0,95.0, 0), v10, z5, tool0;
	MoveL Offs(p0,144.0,95.0, 0), v10, z5, tool0;
	MoveL Offs(p0,145.0,94.0, 0), v10, z5, tool0;
	MoveL Offs(p0,147.0,92.0, 0), v10, z5, tool0;
	MoveL Offs(p0,147.0,91.0, 0), v10, z5, tool0;
	MoveL Offs(p0,147.0,90.0, 0), v10, z5, tool0;
	MoveL Offs(p0,148.0,89.0, 0), v10, z5, tool0;
	MoveL Offs(p0,148.0,88.0, 0), v10, z5, tool0;
	MoveL Offs(p0,149.0,87.0, 0), v10, z5, tool0;
	MoveL Offs(p0,149.0,86.0, 0), v10, z5, tool0;
	MoveL Offs(p0,150.0,83.0, 0), v10, z5, tool0;
	MoveL Offs(p0,152.0,80.0, 0), v10, z5, tool0;
	MoveL Offs(p0,153.0,77.0, 0), v10, z5, tool0;
	MoveL Offs(p0,155.0,74.0, 0), v10, z5, tool0;
	MoveL Offs(p0,157.0,72.0, 0), v10, z5, tool0;
	MoveL Offs(p0,159.0,70.0, 0), v10, z5, tool0;
	MoveL Offs(p0,161.0,68.0, 0), v10, z5, tool0;
	MoveL Offs(p0,163.0,67.0, 0), v10, z5, tool0;
	MoveL Offs(p0,166.0,66.0, 0), v10, z5, tool0;
	MoveL Offs(p0,168.0,65.0, 0), v10, z5, tool0;
	MoveL Offs(p0,171.0,64.0, 0), v10, z5, tool0;
	MoveL Offs(p0,172.0,64.0, 0), v10, z5, tool0;
	MoveL Offs(p0,173.0,64.0, 0), v10, z5, tool0;
	MoveL Offs(p0,175.0,64.0, 0), v10, z5, tool0;
	MoveL Offs(p0,176.0,64.0, 0), v10, z5, tool0;
	MoveL Offs(p0,178.0,64.0, 0), v10, z5, tool0;
	MoveL Offs(p0,179.0,65.0, 0), v10, z5, tool0;
	MoveL Offs(p0,180.0,65.0, 0), v10, z5, tool0;
	MoveL Offs(p0,181.0,65.0, 0), v10, z5, tool0;
	MoveL Offs(p0,183.0,66.0, 0), v10, z5, tool0;
	MoveL Offs(p0,184.0,67.0, 0), v10, z5, tool0;
	MoveL Offs(p0,185.0,68.0, 0), v10, z5, tool0;
	MoveL Offs(p0,185.0,68.0, 0), v10, z5, tool0;
	MoveL Offs(p0,186.0,69.0, 0), v10, z5, tool0;
	MoveL Offs(p0,186.0,70.0, 0), v10, z5, tool0;
	MoveL Offs(p0,187.0,70.0, 0), v10, z5, tool0;
	MoveL Offs(p0,187.0,71.0, 0), v10, z5, tool0;
	MoveL Offs(p0,188.0,74.0, 0), v10, z5, tool0;
	MoveL Offs(p0,188.0,75.0, 0), v10, z5, tool0;
	MoveL Offs(p0,188.0,76.0, 0), v10, z5, tool0;
	MoveL Offs(p0,188.0,77.0, 0), v10, z5, tool0;
	MoveL Offs(p0,188.0,79.0, 0), v10, z5, tool0;
	MoveL Offs(p0,188.0,80.0, 0), v10, z5, tool0;
	MoveL Offs(p0,188.0,81.0, 0), v10, z5, tool0;
	MoveL Offs(p0,187.0,82.0, 0), v10, z5, tool0;
	MoveL Offs(p0,185.0,84.0, 0), v10, z5, tool0;
	MoveL Offs(p0,184.0,86.0, 0), v10, z5, tool0;
	MoveL Offs(p0,183.0,87.0, 0), v10, z5, tool0;
	MoveL Offs(p0,182.0,88.0, 0), v10, z5, tool0;
	MoveL Offs(p0,180.0,89.0, 0), v10, z5, tool0;
	MoveL Offs(p0,179.0,90.0, 0), v10, z5, tool0;
	MoveL Offs(p0,177.0,91.0, 0), v10, z5, tool0;
	MoveL Offs(p0,176.0,92.0, 0), v10, z5, tool0;
	MoveL Offs(p0,174.0,92.0, 0), v10, z5, tool0;
	MoveL Offs(p0,171.0,93.0, 0), v10, z5, tool0;
	MoveL Offs(p0,169.0,93.0, 0), v10, z5, tool0;
	MoveL Offs(p0,168.0,93.0, 0), v10, z5, tool0;
	MoveL Offs(p0,166.0,93.0, 0), v10, z5, tool0;
	MoveL Offs(p0,165.0,92.0, 0), v10, z5, tool0;
	MoveL Offs(p0,164.0,92.0, 0), v10, z5, tool0;
	MoveL Offs(p0,163.0,92.0, 0), v10, z5, tool0;
	MoveL Offs(p0,162.0,91.0, 0), v10, z5, tool0;
	MoveL Offs(p0,162.0,90.0, 0), v10, z5, tool0;
	MoveL Offs(p0,164.0,90.0, 0), v10, z5, tool0;
	MoveL Offs(p0,165.0,90.0, 0), v10, z5, tool0;
	MoveL Offs(p0,166.0,90.0, 0), v10, z5, tool0;
	MoveL Offs(p0,167.0,90.0, 0), v10, z5, tool0;
	MoveL Offs(p0,169.0,90.0, 0), v10, z5, tool0;
	MoveL Offs(p0,170.0,90.0, 0), v10, z5, tool0;
	MoveL Offs(p0,172.0,90.0, 0), v10, z5, tool0;
	MoveL Offs(p0,173.0,89.0, 0), v10, z5, tool0;
	MoveL Offs(p0,174.0,89.0, 0), v10, z5, tool0;
	MoveL Offs(p0,176.0,88.0, 0), v10, z5, tool0;
	MoveL Offs(p0,177.0,88.0, 0), v10, z5, tool0;
	MoveL Offs(p0,178.0,87.0, 0), v10, z5, tool0;
	MoveL Offs(p0,179.0,86.0, 0), v10, z5, tool0;
	MoveL Offs(p0,181.0,83.0, 0), v10, z5, tool0;
	MoveL Offs(p0,182.0,83.0, 0), v10, z5, tool0;
	MoveL Offs(p0,182.0,82.0, 0), v10, z5, tool0;
	MoveL Offs(p0,183.0,81.0, 0), v10, z5, tool0;
	MoveL Offs(p0,183.0,80.0, 0), v10, z5, tool0;
	MoveL Offs(p0,183.0,79.0, 0), v10, z5, tool0;
	MoveL Offs(p0,184.0,79.0, 0), v10, z5, tool0;
	MoveL Offs(p0,184.0,77.0, 0), v10, z5, tool0;
	MoveL Offs(p0,183.0,75.0, 0), v10, z5, tool0;
	MoveL Offs(p0,182.0,73.0, 0), v10, z5, tool0;
	MoveL Offs(p0,181.0,71.0, 0), v10, z5, tool0;
	MoveL Offs(p0,179.0,70.0, 0), v10, z5, tool0;
	MoveL Offs(p0,177.0,69.0, 0), v10, z5, tool0;
	MoveL Offs(p0,174.0,69.0, 0), v10, z5, tool0;
	MoveL Offs(p0,172.0,69.0, 0), v10, z5, tool0;
	MoveL Offs(p0,169.0,69.0, 0), v10, z5, tool0;
	MoveL Offs(p0,166.0,70.0, 0), v10, z5, tool0;
	MoveL Offs(p0,163.0,72.0, 0), v10, z5, tool0;
	MoveL Offs(p0,162.0,73.0, 0), v10, z5, tool0;
	MoveL Offs(p0,160.0,75.0, 0), v10, z5, tool0;
	MoveL Offs(p0,159.0,76.0, 0), v10, z5, tool0;
	MoveL Offs(p0,158.0,78.0, 0), v10, z5, tool0;
	MoveL Offs(p0,157.0,80.0, 0), v10, z5, tool0;
	MoveL Offs(p0,156.0,83.0, 0), v10, z5, tool0;
	MoveL Offs(p0,155.0,85.0, 0), v10, z5, tool0;
	MoveL Offs(p0,154.0,88.0, 0), v10, z5, tool0;
	MoveL Offs(p0,153.0,91.0, 0), v10, z5, tool0;
	MoveL Offs(p0,153.0,92.0, 0), v10, z5, tool0;
	MoveL Offs(p0,152.0,92.0, 0), v10, z5, tool0;
	MoveL Offs(p0,152.0,93.0, 0), v10, z5, tool0;
	MoveL Offs(p0,152.0,94.0, 0), v10, z5, tool0;
	MoveL Offs(p0,151.0,94.0, 0), v10, z5, tool0;
	MoveL Offs(p0,151.0,95.0, 0), v10, z5, tool0;
	MoveL Offs(p0,151.0,95.0, 0), v10, z5, tool0;
	MoveL Offs(p0,149.0,97.0, 0), v10, z5, tool0;
	MoveL Offs(p0,148.0,98.0, 0), v10, z5, tool0;
	MoveL Offs(p0,148.0,99.0, 0), v10, z5, tool0;
	MoveL Offs(p0,147.0,99.0, 0), v10, z5, tool0;
	MoveL Offs(p0,146.0,99.0, 0), v10, z5, tool0;
	MoveL Offs(p0,145.0,100.0, 0), v10, z5, tool0;
	MoveL Offs(p0,145.0,100.0, 0), v10, z5, tool0;
	MoveL Offs(p0,144.0,100.0, 0), v10, z5, tool0;
	MoveL Offs(p0,142.0,101.0, 0), v10, z5, tool0;
	MoveL Offs(p0,141.0,101.0, 0), v10, z5, tool0;
	MoveL Offs(p0,140.0,101.0, 0), v10, z5, tool0;
	MoveL Offs(p0,139.0,101.0, 0), v10, z5, tool0;
	MoveL Offs(p0,138.0,101.0, 0), v10, z5, tool0;
	MoveL Offs(p0,137.0,100.0, 0), v10, z5, tool0;
	MoveL Offs(p0,137.0,100.0, 0), v10, z5, tool0;
	MoveL Offs(p0,136.0,100.0, 0), v10, z5, tool0;
	MoveL Offs(p0,139.0,102.0, 0), v10, z5, tool0;
	MoveL Offs(p0,141.0,102.0, 0), v10, z5, tool0;
	MoveL Offs(p0,143.0,103.0, 0), v10, z5, tool0;
	MoveL Offs(p0,145.0,103.0, 0), v10, z5, tool0;
	MoveL Offs(p0,147.0,103.0, 0), v10, z5, tool0;
	MoveL Offs(p0,149.0,103.0, 0), v10, z5, tool0;
	MoveL Offs(p0,151.0,103.0, 0), v10, z5, tool0;
	MoveL Offs(p0,152.0,103.0, 0), v10, z5, tool0;
	MoveL Offs(p0,155.0,103.0, 0), v10, z5, tool0;
	MoveL Offs(p0,156.0,103.0, 0), v10, z5, tool0;
	MoveL Offs(p0,156.0,103.0, 0), v10, z5, tool0;
	MoveL Offs(p0,157.0,103.0, 0), v10, z5, tool0;
	MoveL Offs(p0,157.0,103.0, 0), v10, z5, tool0;
	MoveL Offs(p0,158.0,103.0, 0), v10, z5, tool0;
	MoveL Offs(p0,158.0,103.0, 0), v10, z5, tool0;
	MoveL Offs(p0,158.0,104.0, 0), v10, z5, tool0;
	MoveL Offs(p0,159.0,104.0, 0), v10, z5, tool0;
	MoveL Offs(p0,160.0,106.0, 0), v10, z5, tool0;
	MoveL Offs(p0,160.0,107.0, 0), v10, z5, tool0;
	MoveL Offs(p0,160.0,107.0, 0), v10, z5, tool0;
	MoveL Offs(p0,160.0,108.0, 0), v10, z5, tool0;
	MoveL Offs(p0,159.0,109.0, 0), v10, z5, tool0;
	MoveL Offs(p0,159.0,109.0, 0), v10, z5, tool0;
	MoveL Offs(p0,158.0,110.0, 0), v10, z5, tool0;
	MoveL Offs(p0,157.0,112.0, 0), v10, z5, tool0;
	MoveL Offs(p0,156.0,113.0, 0), v10, z5, tool0;
	MoveL Offs(p0,156.0,114.0, 0), v10, z5, tool0;
	MoveL Offs(p0,156.0,114.0, 0), v10, z5, tool0;
	MoveL Offs(p0,156.0,115.0, 0), v10, z5, tool0;
	MoveL Offs(p0,156.0,116.0, 0), v10, z5, tool0;
	MoveL Offs(p0,157.0,117.0, 0), v10, z5, tool0;
	MoveL Offs(p0,157.0,118.0, 0), v10, z5, tool0;
	MoveL Offs(p0,159.0,120.0, 0), v10, z5, tool0;
	MoveL Offs(p0,160.0,121.0, 0), v10, z5, tool0;
	MoveL Offs(p0,160.0,121.0, 0), v10, z5, tool0;
	MoveL Offs(p0,161.0,122.0, 0), v10, z5, tool0;
	MoveL Offs(p0,162.0,122.0, 0), v10, z5, tool0;
	MoveL Offs(p0,163.0,123.0, 0), v10, z5, tool0;
	MoveL Offs(p0,165.0,124.0, 0), v10, z5, tool0;
	MoveL Offs(p0,167.0,125.0, 0), v10, z5, tool0;
	MoveL Offs(p0,167.0,125.0, 0), v10, z5, tool0;
	MoveL Offs(p0,168.0,125.0, 0), v10, z5, tool0;
	MoveL Offs(p0,168.0,125.0, 0), v10, z5, tool0;
	MoveL Offs(p0,168.0,126.0, 0), v10, z5, tool0;
	MoveL Offs(p0,169.0,126.0, 0), v10, z5, tool0;
	MoveL Offs(p0,169.0,126.0, 0), v10, z5, tool0;
	MoveL Offs(p0,170.0,128.0, 0), v10, z5, tool0;
	MoveL Offs(p0,170.0,129.0, 0), v10, z5, tool0;
	MoveL Offs(p0,170.0,129.0, 0), v10, z5, tool0;
	MoveL Offs(p0,169.0,130.0, 0), v10, z5, tool0;
	MoveL Offs(p0,169.0,131.0, 0), v10, z5, tool0;
	MoveL Offs(p0,169.0,132.0, 0), v10, z5, tool0;
	MoveL Offs(p0,168.0,133.0, 0), v10, z5, tool0;
	MoveL Offs(p0,167.0,135.0, 0), v10, z5, tool0;
	MoveL Offs(p0,167.0,136.0, 0), v10, z5, tool0;
	MoveL Offs(p0,166.0,137.0, 0), v10, z5, tool0;
	MoveL Offs(p0,166.0,138.0, 0), v10, z5, tool0;
	MoveL Offs(p0,166.0,139.0, 0), v10, z5, tool0;
	MoveL Offs(p0,166.0,140.0, 0), v10, z5, tool0;
	MoveL Offs(p0,166.0,141.0, 0), v10, z5, tool0;
	MoveL Offs(p0,166.0,142.0, 0), v10, z5, tool0;
	MoveL Offs(p0,166.0,145.0, 0), v10, z5, tool0;
	MoveL Offs(p0,167.0,146.0, 0), v10, z5, tool0;
	MoveL Offs(p0,167.0,148.0, 0), v10, z5, tool0;
	MoveL Offs(p0,167.0,149.0, 0), v10, z5, tool0;
	MoveL Offs(p0,168.0,149.0, 0), v10, z5, tool0;
	MoveL Offs(p0,168.0,150.0, 0), v10, z5, tool0;
	MoveL Offs(p0,169.0,151.0, 0), v10, z5, tool0;
	MoveL Offs(p0,170.0,152.0, 0), v10, z5, tool0;
	MoveL Offs(p0,170.0,152.0, 0), v10, z5, tool0;
	MoveL Offs(p0,172.0,154.0, 0), v10, z5, tool0;
	MoveL Offs(p0,172.0,154.0, 0), v10, z5, tool0;
	MoveL Offs(p0,172.0,155.0, 0), v10, z5, tool0;
	MoveL Offs(p0,172.0,155.0, 0), v10, z5, tool0;
	MoveL Offs(p0,172.0,156.0, 0), v10, z5, tool0;
	MoveL Offs(p0,170.0,157.0, 0), v10, z5, tool0;
	MoveL Offs(p0,170.0,157.0, 0), v10, z5, tool0;
	MoveL Offs(p0,167.0,156.0, 0), v10, z5, tool0;
	MoveL Offs(p0,166.0,155.0, 0), v10, z5, tool0;
	MoveL Offs(p0,164.0,154.0, 0), v10, z5, tool0;
	MoveL Offs(p0,161.0,153.0, 0), v10, z5, tool0;
	MoveL Offs(p0,159.0,151.0, 0), v10, z5, tool0;
	MoveL Offs(p0,156.0,149.0, 0), v10, z5, tool0;
	MoveL Offs(p0,153.0,147.0, 0), v10, z5, tool0;
	MoveL Offs(p0,150.0,144.0, 0), v10, z5, tool0;
	MoveL Offs(p0,147.0,142.0, 0), v10, z5, tool0;
	MoveL Offs(p0,142.0,138.0, 0), v10, z5, tool0;
	MoveL Offs(p0,141.0,139.0, 0), v10, z5, tool0;
	MoveL Offs(p0,141.0,141.0, 0), v10, z5, tool0;
	MoveL Offs(p0,140.0,142.0, 0), v10, z5, tool0;
	MoveL Offs(p0,140.0,142.0, 0), v10, z5, tool0;
	MoveL Offs(p0,139.0,142.0, 0), v10, z5, tool0;
	MoveL Offs(p0,138.0,142.0, 0), v10, z5, tool0;
	MoveL Offs(p0,138.0,142.0, 0), v10, z5, tool0;
	MoveL Offs(p0,137.0,142.0, 0), v10, z5, tool0;
	MoveL Offs(p0,136.0,142.0, 0), v10, z5, tool0;
	MoveL Offs(p0,135.0,144.0, 0), v10, z5, tool0;
	MoveL Offs(p0,135.0,144.0, 0), v10, z5, tool0;
	MoveL Offs(p0,134.0,145.0, 0), v10, z5, tool0;
	MoveL Offs(p0,134.0,145.0, 0), v10, z5, tool0;
	MoveL Offs(p0,134.0,145.0, 0), v10, z5, tool0;
	MoveL Offs(p0,134.0,145.0, 0), v10, z5, tool0;
	MoveL Offs(p0,132.0,145.0, 0), v10, z5, tool0;
	MoveL Offs(p0,131.0,144.0, 0), v10, z5, tool0;
	MoveL Offs(p0,130.0,144.0, 0), v10, z5, tool0;
	MoveL Offs(p0,129.0,144.0, 0), v10, z5, tool0;
	MoveL Offs(p0,129.0,144.0, 0), v10, z5, tool0;
	MoveL Offs(p0,128.0,143.0, 0), v10, z5, tool0;
	MoveL Offs(p0,125.0,142.0, 0), v10, z5, tool0;
	MoveL Offs(p0,124.0,142.0, 0), v10, z5, tool0;
	MoveL Offs(p0,124.0,142.0, 0), v10, z5, tool0;
	MoveL Offs(p0,123.0,142.0, 0), v10, z5, tool0;
	MoveL Offs(p0,123.0,141.0, 0), v10, z5, tool0;
	MoveL Offs(p0,123.0,141.0, 0), v10, z5, tool0;
	MoveL Offs(p0,122.0,141.0, 0), v10, z5, tool0;
	MoveL Offs(p0,122.0,141.0, 0), v10, z5, tool0;
	MoveL Offs(p0,123.0,144.0, 0), v10, z5, tool0;
	MoveL Offs(p0,124.0,145.0, 0), v10, z5, tool0;
	MoveL Offs(p0,124.0,146.0, 0), v10, z5, tool0;
	MoveL Offs(p0,125.0,147.0, 0), v10, z5, tool0;
	MoveL Offs(p0,125.0,148.0, 0), v10, z5, tool0;
	MoveL Offs(p0,127.0,150.0, 0), v10, z5, tool0;
	MoveL Offs(p0,127.0,151.0, 0), v10, z5, tool0;
	MoveL Offs(p0,128.0,152.0, 0), v10, z5, tool0;
	MoveL Offs(p0,128.0,153.0, 0), v10, z5, tool0;
	MoveL Offs(p0,128.0,153.0, 0), v10, z5, tool0;
	MoveL Offs(p0,129.0,154.0, 0), v10, z5, tool0;
	MoveL Offs(p0,129.0,155.0, 0), v10, z5, tool0;
	MoveL Offs(p0,129.0,155.0, 0), v10, z5, tool0;
	MoveL Offs(p0,129.0,155.0, 0), v10, z5, tool0;
	MoveL Offs(p0,128.0,158.0, 0), v10, z5, tool0;
	MoveL Offs(p0,128.0,158.0, 0), v10, z5, tool0;
	MoveL Offs(p0,127.0,158.0, 0), v10, z5, tool0;
	MoveL Offs(p0,127.0,158.0, 0), v10, z5, tool0;
	MoveL Offs(p0,126.0,158.0, 0), v10, z5, tool0;
	MoveL Offs(p0,125.0,158.0, 0), v10, z5, tool0;
	MoveL Offs(p0,125.0,158.0, 0), v10, z5, tool0;
	MoveL Offs(p0,123.0,156.0, 0), v10, z5, tool0;
	MoveL Offs(p0,122.0,155.0, 0), v10, z5, tool0;
	MoveL Offs(p0,121.0,154.0, 0), v10, z5, tool0;
	MoveL Offs(p0,121.0,153.0, 0), v10, z5, tool0;
	MoveL Offs(p0,120.0,152.0, 0), v10, z5, tool0;
	MoveL Offs(p0,118.0,150.0, 0), v10, z5, tool0;
	MoveL Offs(p0,118.0,149.0, 0), v10, z5, tool0;
	MoveL Offs(p0,117.0,149.0, 0), v10, z5, tool0;
	MoveL Offs(p0,117.0,148.0, 0), v10, z5, tool0;
	MoveL Offs(p0,116.0,148.0, 0), v10, z5, tool0;
	MoveL Offs(p0,116.0,148.0, 0), v10, z5, tool0;
	MoveL Offs(p0,116.0,147.0, 0), v10, z5, tool0;
	MoveL Offs(p0,115.0,147.0, 0), v10, z5, tool0;
	MoveL Offs(p0,115.0,147.0, 0), v10, z5, tool0;
	MoveL Offs(p0,112.0,147.0, 0), v10, z5, tool0;
	MoveL Offs(p0,111.0,146.0, 0), v10, z5, tool0;
	MoveL Offs(p0,109.0,146.0, 0), v10, z5, tool0;
	MoveL Offs(p0,108.0,146.0, 0), v10, z5, tool0;
	MoveL Offs(p0,107.0,147.0, 0), v10, z5, tool0;
	MoveL Offs(p0,105.0,147.0, 0), v10, z5, tool0;
	MoveL Offs(p0,104.0,147.0, 0), v10, z5, tool0;
	MoveL Offs(p0,102.0,148.0, 0), v10, z5, tool0;
	MoveL Offs(p0,100.0,148.0, 0), v10, z5, tool0;
	MoveL Offs(p0,98.0,149.0, 0), v10, z5, tool0;
	MoveL Offs(p0,97.0,149.0, 0), v10, z5, tool0;
	MoveL Offs(p0,96.0,149.0, 0), v10, z5, tool0;
	MoveL Offs(p0,95.0,150.0, 0), v10, z5, tool0;
	MoveL Offs(p0,95.0,150.0, 0), v10, z5, tool0;
	MoveL Offs(p0,94.0,150.0, 0), v10, z5, tool0;
	MoveL Offs(p0,93.0,150.0, 0), v10, z5, tool0;
	MoveL Offs(p0,92.0,150.0, 0), v10, z5, tool0;
	MoveL Offs(p0,89.0,150.0, 0), v10, z5, tool0;
	MoveL Offs(p0,89.0,154.0, 0), v10, z5, tool0;
	MoveL Offs(p0,88.0,157.0, 0), v10, z5, tool0;
	MoveL Offs(p0,88.0,158.0, 0), v10, z5, tool0;
	MoveL Offs(p0,88.0,160.0, 0), v10, z5, tool0;
	MoveL Offs(p0,87.0,162.0, 0), v10, z5, tool0;
	MoveL Offs(p0,87.0,164.0, 0), v10, z5, tool0;
	MoveL Offs(p0,87.0,165.0, 0), v10, z5, tool0;
	MoveL Offs(p0,86.0,167.0, 0), v10, z5, tool0;
	MoveL Offs(p0,86.0,168.0, 0), v10, z5, tool0;
	MoveL Offs(p0,86.0,169.0, 0), v10, z5, tool0;
	MoveL Offs(p0,85.0,171.0, 0), v10, z5, tool0;
	MoveL Offs(p0,84.0,171.0, 0), v10, z5, tool0;
	MoveL Offs(p0,84.0,171.0, 0), v10, z5, tool0;
	MoveL Offs(p0,84.0,171.0, 0), v10, z5, tool0;
	MoveL Offs(p0,83.0,171.0, 0), v10, z5, tool0;
	MoveL Offs(p0,83.0,172.0, 0), v10, z5, tool0;
	MoveL Offs(p0,81.0,172.0, 0), v10, z5, tool0;
	MoveL Offs(p0,82.0,168.0, 0), v10, z5, tool0;
	MoveL Offs(p0,82.0,164.0, 0), v10, z5, tool0;
	MoveL Offs(p0,81.0,167.0, 0), v10, z5, tool0;
	MoveL Offs(p0,79.0,170.0, 0), v10, z5, tool0;
	MoveL Offs(p0,78.0,172.0, 0), v10, z5, tool0;
	MoveL Offs(p0,77.0,174.0, 0), v10, z5, tool0;
	MoveL Offs(p0,77.0,176.0, 0), v10, z5, tool0;
	MoveL Offs(p0,76.0,178.0, 0), v10, z5, tool0;
	MoveL Offs(p0,75.0,179.0, 0), v10, z5, tool0;
	MoveL Offs(p0,74.0,181.0, 0), v10, z5, tool0;
	MoveL Offs(p0,73.0,182.0, 0), v10, z5, tool0;
	MoveL Offs(p0,73.0,183.0, 0), v10, z5, tool0;
	MoveL Offs(p0,71.0,186.0, 0), v10, z5, tool0;
	MoveL Offs(p0,70.0,186.0, 0), v10, z5, tool0;
	MoveL Offs(p0,70.0,187.0, 0), v10, z5, tool0;
	MoveL Offs(p0,69.0,187.0, 0), v10, z5, tool0;
	MoveL Offs(p0,69.0,187.0, 0), v10, z5, tool0;
	MoveL Offs(p0,68.0,187.0, 0), v10, z5, tool0;
	MoveL Offs(p0,68.0,188.0, 0), v10, z5, tool0;
	MoveL Offs(p0,67.0,188.0, 0), v10, z5, tool0;
	MoveL Offs(p0,65.0,187.0, 0), v10, z5, tool0;
	MoveJ Offs(p0,65.0,187.0, 20), v10, z1, tool0;
	MoveJ Offs(p0,69.0,186.0, 20), v10, z1, tool0;
	MoveJ Offs(p0,69.0,186.0, 0), v10, z1, tool0;
	MoveL Offs(p0,71.0,184.0, 0), v10, z5, tool0;
	MoveL Offs(p0,72.0,183.0, 0), v10, z5, tool0;
	MoveL Offs(p0,72.0,182.0, 0), v10, z5, tool0;
	MoveL Offs(p0,73.0,181.0, 0), v10, z5, tool0;
	MoveL Offs(p0,74.0,179.0, 0), v10, z5, tool0;
	MoveL Offs(p0,74.0,178.0, 0), v10, z5, tool0;
	MoveL Offs(p0,75.0,177.0, 0), v10, z5, tool0;
	MoveL Offs(p0,76.0,175.0, 0), v10, z5, tool0;
	MoveL Offs(p0,77.0,173.0, 0), v10, z5, tool0;
	MoveL Offs(p0,78.0,170.0, 0), v10, z5, tool0;
	MoveL Offs(p0,79.0,168.0, 0), v10, z5, tool0;
	MoveL Offs(p0,80.0,166.0, 0), v10, z5, tool0;
	MoveL Offs(p0,80.0,164.0, 0), v10, z5, tool0;
	MoveL Offs(p0,81.0,162.0, 0), v10, z5, tool0;
	MoveL Offs(p0,81.0,161.0, 0), v10, z5, tool0;
	MoveL Offs(p0,81.0,160.0, 0), v10, z5, tool0;
	MoveL Offs(p0,81.0,159.0, 0), v10, z5, tool0;
	MoveL Offs(p0,83.0,161.0, 0), v10, z5, tool0;
	MoveL Offs(p0,83.0,162.0, 0), v10, z5, tool0;
	MoveL Offs(p0,83.0,163.0, 0), v10, z5, tool0;
	MoveL Offs(p0,83.0,164.0, 0), v10, z5, tool0;
	MoveL Offs(p0,83.0,166.0, 0), v10, z5, tool0;
	MoveL Offs(p0,83.0,168.0, 0), v10, z5, tool0;
	MoveL Offs(p0,83.0,169.0, 0), v10, z5, tool0;
	MoveL Offs(p0,83.0,169.0, 0), v10, z5, tool0;
	MoveL Offs(p0,83.0,170.0, 0), v10, z5, tool0;
	MoveL Offs(p0,83.0,170.0, 0), v10, z5, tool0;
	MoveL Offs(p0,83.0,171.0, 0), v10, z5, tool0;
	MoveL Offs(p0,83.0,171.0, 0), v10, z5, tool0;
	MoveL Offs(p0,83.0,171.0, 0), v10, z5, tool0;
	MoveL Offs(p0,83.0,171.0, 0), v10, z5, tool0;
	MoveL Offs(p0,85.0,168.0, 0), v10, z5, tool0;
	MoveL Offs(p0,85.0,167.0, 0), v10, z5, tool0;
	MoveL Offs(p0,85.0,166.0, 0), v10, z5, tool0;
	MoveL Offs(p0,86.0,165.0, 0), v10, z5, tool0;
	MoveL Offs(p0,86.0,164.0, 0), v10, z5, tool0;
	MoveL Offs(p0,86.0,161.0, 0), v10, z5, tool0;
	MoveL Offs(p0,87.0,159.0, 0), v10, z5, tool0;
	MoveL Offs(p0,87.0,157.0, 0), v10, z5, tool0;
	MoveL Offs(p0,87.0,156.0, 0), v10, z5, tool0;
	MoveL Offs(p0,87.0,154.0, 0), v10, z5, tool0;
	MoveL Offs(p0,87.0,153.0, 0), v10, z5, tool0;
	MoveL Offs(p0,88.0,152.0, 0), v10, z5, tool0;
	MoveL Offs(p0,88.0,151.0, 0), v10, z5, tool0;
	MoveL Offs(p0,88.0,150.0, 0), v10, z5, tool0;
	MoveL Offs(p0,85.0,153.0, 0), v10, z5, tool0;
	MoveL Offs(p0,85.0,153.0, 0), v10, z5, tool0;
	MoveL Offs(p0,84.0,154.0, 0), v10, z5, tool0;
	MoveL Offs(p0,83.0,155.0, 0), v10, z5, tool0;
	MoveL Offs(p0,82.0,156.0, 0), v10, z5, tool0;
	MoveL Offs(p0,81.0,158.0, 0), v10, z5, tool0;
	MoveL Offs(p0,79.0,160.0, 0), v10, z5, tool0;
	MoveL Offs(p0,78.0,161.0, 0), v10, z5, tool0;
	MoveL Offs(p0,77.0,163.0, 0), v10, z5, tool0;
	MoveL Offs(p0,77.0,163.0, 0), v10, z5, tool0;
	MoveL Offs(p0,76.0,164.0, 0), v10, z5, tool0;
	MoveL Offs(p0,76.0,164.0, 0), v10, z5, tool0;
	MoveL Offs(p0,75.0,165.0, 0), v10, z5, tool0;
	MoveL Offs(p0,75.0,165.0, 0), v10, z5, tool0;
	MoveL Offs(p0,75.0,165.0, 0), v10, z5, tool0;
	MoveL Offs(p0,73.0,163.0, 0), v10, z5, tool0;
	MoveL Offs(p0,73.0,163.0, 0), v10, z5, tool0;
	MoveL Offs(p0,74.0,161.0, 0), v10, z5, tool0;
	MoveL Offs(p0,74.0,160.0, 0), v10, z5, tool0;
	MoveL Offs(p0,75.0,158.0, 0), v10, z5, tool0;
	MoveL Offs(p0,75.0,157.0, 0), v10, z5, tool0;
	MoveL Offs(p0,76.0,155.0, 0), v10, z5, tool0;
	MoveL Offs(p0,77.0,153.0, 0), v10, z5, tool0;
	MoveL Offs(p0,79.0,150.0, 0), v10, z5, tool0;
	MoveL Offs(p0,80.0,148.0, 0), v10, z5, tool0;
	MoveL Offs(p0,81.0,146.0, 0), v10, z5, tool0;
	MoveL Offs(p0,82.0,144.0, 0), v10, z5, tool0;
	MoveL Offs(p0,82.0,142.0, 0), v10, z5, tool0;
	MoveL Offs(p0,83.0,141.0, 0), v10, z5, tool0;
	MoveL Offs(p0,83.0,140.0, 0), v10, z5, tool0;
	MoveL Offs(p0,84.0,140.0, 0), v10, z5, tool0;
	MoveL Offs(p0,84.0,139.0, 0), v10, z5, tool0;
	MoveL Offs(p0,84.0,139.0, 0), v10, z5, tool0;
	MoveL Offs(p0,84.0,139.0, 0), v10, z5, tool0;
	MoveL Offs(p0,80.0,141.0, 0), v10, z5, tool0;
	MoveL Offs(p0,79.0,142.0, 0), v10, z5, tool0;
	MoveL Offs(p0,79.0,142.0, 0), v10, z5, tool0;
	MoveL Offs(p0,78.0,142.0, 0), v10, z5, tool0;
	MoveL Offs(p0,78.0,143.0, 0), v10, z5, tool0;
	MoveL Offs(p0,77.0,143.0, 0), v10, z5, tool0;
	MoveL Offs(p0,76.0,143.0, 0), v10, z5, tool0;
	MoveL Offs(p0,75.0,145.0, 0), v10, z5, tool0;
	MoveL Offs(p0,75.0,146.0, 0), v10, z5, tool0;
	MoveL Offs(p0,74.0,146.0, 0), v10, z5, tool0;
	MoveL Offs(p0,73.0,148.0, 0), v10, z5, tool0;
	MoveL Offs(p0,73.0,150.0, 0), v10, z5, tool0;
	MoveL Offs(p0,72.0,151.0, 0), v10, z5, tool0;
	MoveL Offs(p0,71.0,152.0, 0), v10, z5, tool0;
	MoveL Offs(p0,71.0,153.0, 0), v10, z5, tool0;
	MoveL Offs(p0,70.0,154.0, 0), v10, z5, tool0;
	MoveL Offs(p0,69.0,156.0, 0), v10, z5, tool0;
	MoveL Offs(p0,68.0,157.0, 0), v10, z5, tool0;
	MoveL Offs(p0,67.0,159.0, 0), v10, z5, tool0;
	MoveL Offs(p0,66.0,161.0, 0), v10, z5, tool0;
	MoveL Offs(p0,66.0,162.0, 0), v10, z5, tool0;
	MoveL Offs(p0,65.0,163.0, 0), v10, z5, tool0;
	MoveL Offs(p0,65.0,163.0, 0), v10, z5, tool0;
	MoveL Offs(p0,65.0,164.0, 0), v10, z5, tool0;
	MoveL Offs(p0,65.0,164.0, 0), v10, z5, tool0;
	MoveL Offs(p0,65.0,164.0, 0), v10, z5, tool0;
	MoveL Offs(p0,65.0,164.0, 0), v10, z5, tool0;
	MoveL Offs(p0,67.0,164.0, 0), v10, z5, tool0;
	MoveL Offs(p0,67.0,163.0, 0), v10, z5, tool0;
	MoveL Offs(p0,67.0,163.0, 0), v10, z5, tool0;
	MoveL Offs(p0,68.0,163.0, 0), v10, z5, tool0;
	MoveL Offs(p0,71.0,164.0, 0), v10, z5, tool0;
	MoveL Offs(p0,71.0,166.0, 0), v10, z5, tool0;
	MoveL Offs(p0,70.0,169.0, 0), v10, z5, tool0;
	MoveL Offs(p0,70.0,172.0, 0), v10, z5, tool0;
	MoveL Offs(p0,69.0,175.0, 0), v10, z5, tool0;
	MoveL Offs(p0,69.0,178.0, 0), v10, z5, tool0;
	MoveL Offs(p0,68.0,180.0, 0), v10, z5, tool0;
	MoveL Offs(p0,67.0,183.0, 0), v10, z5, tool0;
	MoveL Offs(p0,67.0,184.0, 0), v10, z5, tool0;
	MoveL Offs(p0,66.0,186.0, 0), v10, z5, tool0;
	MoveL Offs(p0,66.0,186.0, 0), v10, z5, tool0;
	MoveL Offs(p0,68.0,187.0, 0), v10, z5, tool0;
	MoveL Offs(p0,68.0,186.0, 0), v10, z5, tool0;
	MoveL Offs(p0,69.0,186.0, 0), v10, z5, tool0;
	MoveL Offs(p0,69.0,186.0, 0), v10, z5, tool0;
	MoveJ Offs(p0,69.0,186.0, 20), v10, z1, tool0;
	MoveJ Offs(p0,50.0,157.0, 20), v10, z1, tool0;
	MoveJ Offs(p0,50.0,157.0, 0), v10, z1, tool0;
	MoveL Offs(p0,53.0,156.0, 0), v10, z5, tool0;
	MoveL Offs(p0,53.0,156.0, 0), v10, z5, tool0;
	MoveL Offs(p0,54.0,155.0, 0), v10, z5, tool0;
	MoveL Offs(p0,55.0,155.0, 0), v10, z5, tool0;
	MoveL Offs(p0,56.0,154.0, 0), v10, z5, tool0;
	MoveL Offs(p0,56.0,154.0, 0), v10, z5, tool0;
	MoveL Offs(p0,57.0,154.0, 0), v10, z5, tool0;
	MoveL Offs(p0,59.0,152.0, 0), v10, z5, tool0;
	MoveL Offs(p0,59.0,152.0, 0), v10, z5, tool0;
	MoveL Offs(p0,60.0,151.0, 0), v10, z5, tool0;
	MoveL Offs(p0,60.0,151.0, 0), v10, z5, tool0;
	MoveL Offs(p0,60.0,151.0, 0), v10, z5, tool0;
	MoveL Offs(p0,60.0,151.0, 0), v10, z5, tool0;
	MoveL Offs(p0,60.0,151.0, 0), v10, z5, tool0;
	MoveL Offs(p0,60.0,150.0, 0), v10, z5, tool0;
	MoveL Offs(p0,61.0,152.0, 0), v10, z5, tool0;
	MoveL Offs(p0,61.0,153.0, 0), v10, z5, tool0;
	MoveL Offs(p0,61.0,153.0, 0), v10, z5, tool0;
	MoveL Offs(p0,61.0,155.0, 0), v10, z5, tool0;
	MoveL Offs(p0,61.0,155.0, 0), v10, z5, tool0;
	MoveL Offs(p0,61.0,156.0, 0), v10, z5, tool0;
	MoveL Offs(p0,61.0,156.0, 0), v10, z5, tool0;
	MoveL Offs(p0,61.0,156.0, 0), v10, z5, tool0;
	MoveL Offs(p0,63.0,154.0, 0), v10, z5, tool0;
	MoveL Offs(p0,64.0,152.0, 0), v10, z5, tool0;
	MoveL Offs(p0,65.0,151.0, 0), v10, z5, tool0;
	MoveL Offs(p0,66.0,150.0, 0), v10, z5, tool0;
	MoveL Offs(p0,67.0,148.0, 0), v10, z5, tool0;
	MoveL Offs(p0,68.0,147.0, 0), v10, z5, tool0;
	MoveL Offs(p0,69.0,146.0, 0), v10, z5, tool0;
	MoveL Offs(p0,70.0,144.0, 0), v10, z5, tool0;
	MoveL Offs(p0,67.0,141.0, 0), v10, z5, tool0;
	MoveL Offs(p0,64.0,139.0, 0), v10, z5, tool0;
	MoveL Offs(p0,64.0,139.0, 0), v10, z5, tool0;
	MoveL Offs(p0,64.0,139.0, 0), v10, z5, tool0;
	MoveL Offs(p0,63.0,138.0, 0), v10, z5, tool0;
	MoveL Offs(p0,63.0,138.0, 0), v10, z5, tool0;
	MoveL Offs(p0,63.0,138.0, 0), v10, z5, tool0;
	MoveL Offs(p0,63.0,138.0, 0), v10, z5, tool0;
	MoveL Offs(p0,59.0,141.0, 0), v10, z5, tool0;
	MoveL Offs(p0,58.0,142.0, 0), v10, z5, tool0;
	MoveL Offs(p0,57.0,142.0, 0), v10, z5, tool0;
	MoveL Offs(p0,56.0,143.0, 0), v10, z5, tool0;
	MoveL Offs(p0,55.0,143.0, 0), v10, z5, tool0;
	MoveL Offs(p0,55.0,144.0, 0), v10, z5, tool0;
	MoveL Offs(p0,55.0,144.0, 0), v10, z5, tool0;
	MoveL Offs(p0,54.0,144.0, 0), v10, z5, tool0;
	MoveL Offs(p0,54.0,144.0, 0), v10, z5, tool0;
	MoveL Offs(p0,56.0,148.0, 0), v10, z5, tool0;
	MoveL Offs(p0,55.0,149.0, 0), v10, z5, tool0;
	MoveL Offs(p0,54.0,150.0, 0), v10, z5, tool0;
	MoveL Offs(p0,53.0,151.0, 0), v10, z5, tool0;
	MoveL Offs(p0,52.0,152.0, 0), v10, z5, tool0;
	MoveL Offs(p0,51.0,154.0, 0), v10, z5, tool0;
	MoveL Offs(p0,49.0,155.0, 0), v10, z5, tool0;
	MoveL Offs(p0,47.0,158.0, 0), v10, z5, tool0;
	MoveL Offs(p0,47.0,158.0, 0), v10, z5, tool0;
	MoveL Offs(p0,47.0,158.0, 0), v10, z5, tool0;
	MoveL Offs(p0,47.0,158.0, 0), v10, z5, tool0;
	MoveL Offs(p0,47.0,159.0, 0), v10, z5, tool0;
	MoveL Offs(p0,47.0,159.0, 0), v10, z5, tool0;
	MoveL Offs(p0,48.0,159.0, 0), v10, z5, tool0;
	MoveL Offs(p0,50.0,158.0, 0), v10, z5, tool0;
	MoveL Offs(p0,50.0,158.0, 0), v10, z5, tool0;
	MoveL Offs(p0,50.0,157.0, 0), v10, z5, tool0;
	MoveL Offs(p0,50.0,157.0, 0), v10, z5, tool0;
	MoveJ Offs(p0,50.0,157.0, 20), v10, z1, tool0;
	MoveJ Offs(p0,170.0,156.0, 20), v10, z1, tool0;
	MoveJ Offs(p0,170.0,156.0, 0), v10, z1, tool0;
	MoveL Offs(p0,171.0,154.0, 0), v10, z5, tool0;
	MoveL Offs(p0,168.0,152.0, 0), v10, z5, tool0;
	MoveL Offs(p0,168.0,152.0, 0), v10, z5, tool0;
	MoveL Offs(p0,167.0,152.0, 0), v10, z5, tool0;
	MoveL Offs(p0,164.0,150.0, 0), v10, z5, tool0;
	MoveL Offs(p0,161.0,147.0, 0), v10, z5, tool0;
	MoveL Offs(p0,157.0,144.0, 0), v10, z5, tool0;
	MoveL Offs(p0,153.0,141.0, 0), v10, z5, tool0;
	MoveL Offs(p0,149.0,137.0, 0), v10, z5, tool0;
	MoveL Offs(p0,145.0,134.0, 0), v10, z5, tool0;
	MoveL Offs(p0,141.0,130.0, 0), v10, z5, tool0;
	MoveL Offs(p0,138.0,127.0, 0), v10, z5, tool0;
	MoveL Offs(p0,136.0,125.0, 0), v10, z5, tool0;
	MoveL Offs(p0,134.0,122.0, 0), v10, z5, tool0;
	MoveL Offs(p0,133.0,125.0, 0), v10, z5, tool0;
	MoveL Offs(p0,134.0,126.0, 0), v10, z5, tool0;
	MoveL Offs(p0,135.0,128.0, 0), v10, z5, tool0;
	MoveL Offs(p0,136.0,129.0, 0), v10, z5, tool0;
	MoveL Offs(p0,137.0,131.0, 0), v10, z5, tool0;
	MoveL Offs(p0,138.0,133.0, 0), v10, z5, tool0;
	MoveL Offs(p0,139.0,134.0, 0), v10, z5, tool0;
	MoveL Offs(p0,141.0,135.0, 0), v10, z5, tool0;
	MoveL Offs(p0,142.0,137.0, 0), v10, z5, tool0;
	MoveL Offs(p0,144.0,139.0, 0), v10, z5, tool0;
	MoveL Offs(p0,145.0,139.0, 0), v10, z5, tool0;
	MoveL Offs(p0,146.0,140.0, 0), v10, z5, tool0;
	MoveL Offs(p0,147.0,141.0, 0), v10, z5, tool0;
	MoveL Offs(p0,148.0,141.0, 0), v10, z5, tool0;
	MoveL Offs(p0,149.0,142.0, 0), v10, z5, tool0;
	MoveL Offs(p0,149.0,142.0, 0), v10, z5, tool0;
	MoveL Offs(p0,149.0,142.0, 0), v10, z5, tool0;
	MoveL Offs(p0,150.0,142.0, 0), v10, z5, tool0;
	MoveL Offs(p0,152.0,144.0, 0), v10, z5, tool0;
	MoveL Offs(p0,152.0,144.0, 0), v10, z5, tool0;
	MoveL Offs(p0,153.0,145.0, 0), v10, z5, tool0;
	MoveL Offs(p0,153.0,145.0, 0), v10, z5, tool0;
	MoveL Offs(p0,157.0,148.0, 0), v10, z5, tool0;
	MoveL Offs(p0,157.0,148.0, 0), v10, z5, tool0;
	MoveL Offs(p0,158.0,149.0, 0), v10, z5, tool0;
	MoveL Offs(p0,158.0,149.0, 0), v10, z5, tool0;
	MoveL Offs(p0,159.0,150.0, 0), v10, z5, tool0;
	MoveL Offs(p0,160.0,150.0, 0), v10, z5, tool0;
	MoveL Offs(p0,162.0,152.0, 0), v10, z5, tool0;
	MoveL Offs(p0,162.0,152.0, 0), v10, z5, tool0;
	MoveL Offs(p0,162.0,152.0, 0), v10, z5, tool0;
	MoveL Offs(p0,162.0,152.0, 0), v10, z5, tool0;
	MoveL Offs(p0,165.0,154.0, 0), v10, z5, tool0;
	MoveL Offs(p0,166.0,154.0, 0), v10, z5, tool0;
	MoveL Offs(p0,167.0,155.0, 0), v10, z5, tool0;
	MoveL Offs(p0,168.0,156.0, 0), v10, z5, tool0;
	MoveL Offs(p0,169.0,156.0, 0), v10, z5, tool0;
	MoveL Offs(p0,169.0,156.0, 0), v10, z5, tool0;
	MoveL Offs(p0,170.0,156.0, 0), v10, z5, tool0;
	MoveL Offs(p0,170.0,156.0, 0), v10, z5, tool0;
	MoveJ Offs(p0,170.0,156.0, 20), v10, z1, tool0;
	MoveJ Offs(p0,166.0,148.0, 20), v10, z1, tool0;
	MoveJ Offs(p0,166.0,148.0, 0), v10, z1, tool0;
	MoveL Offs(p0,165.0,145.0, 0), v10, z5, tool0;
	MoveL Offs(p0,165.0,143.0, 0), v10, z5, tool0;
	MoveL Offs(p0,165.0,142.0, 0), v10, z5, tool0;
	MoveL Offs(p0,165.0,140.0, 0), v10, z5, tool0;
	MoveL Offs(p0,165.0,138.0, 0), v10, z5, tool0;
	MoveL Offs(p0,165.0,137.0, 0), v10, z5, tool0;
	MoveL Offs(p0,166.0,135.0, 0), v10, z5, tool0;
	MoveL Offs(p0,166.0,134.0, 0), v10, z5, tool0;
	MoveL Offs(p0,167.0,132.0, 0), v10, z5, tool0;
	MoveL Offs(p0,168.0,130.0, 0), v10, z5, tool0;
	MoveL Offs(p0,168.0,129.0, 0), v10, z5, tool0;
	MoveL Offs(p0,168.0,129.0, 0), v10, z5, tool0;
	MoveL Offs(p0,168.0,128.0, 0), v10, z5, tool0;
	MoveL Offs(p0,168.0,128.0, 0), v10, z5, tool0;
	MoveL Offs(p0,168.0,127.0, 0), v10, z5, tool0;
	MoveL Offs(p0,168.0,127.0, 0), v10, z5, tool0;
	MoveL Offs(p0,168.0,127.0, 0), v10, z5, tool0;
	MoveL Offs(p0,166.0,125.0, 0), v10, z5, tool0;
	MoveL Offs(p0,165.0,125.0, 0), v10, z5, tool0;
	MoveL Offs(p0,164.0,125.0, 0), v10, z5, tool0;
	MoveL Offs(p0,163.0,124.0, 0), v10, z5, tool0;
	MoveL Offs(p0,162.0,124.0, 0), v10, z5, tool0;
	MoveL Offs(p0,161.0,123.0, 0), v10, z5, tool0;
	MoveL Offs(p0,160.0,123.0, 0), v10, z5, tool0;
	MoveL Offs(p0,156.0,122.0, 0), v10, z5, tool0;
	MoveL Offs(p0,154.0,121.0, 0), v10, z5, tool0;
	MoveL Offs(p0,152.0,121.0, 0), v10, z5, tool0;
	MoveL Offs(p0,150.0,120.0, 0), v10, z5, tool0;
	MoveL Offs(p0,148.0,119.0, 0), v10, z5, tool0;
	MoveL Offs(p0,147.0,118.0, 0), v10, z5, tool0;
	MoveL Offs(p0,145.0,117.0, 0), v10, z5, tool0;
	MoveL Offs(p0,143.0,116.0, 0), v10, z5, tool0;
	MoveL Offs(p0,142.0,116.0, 0), v10, z5, tool0;
	MoveL Offs(p0,140.0,114.0, 0), v10, z5, tool0;
	MoveL Offs(p0,140.0,114.0, 0), v10, z5, tool0;
	MoveL Offs(p0,139.0,114.0, 0), v10, z5, tool0;
	MoveL Offs(p0,139.0,114.0, 0), v10, z5, tool0;
	MoveL Offs(p0,139.0,115.0, 0), v10, z5, tool0;
	MoveL Offs(p0,137.0,115.0, 0), v10, z5, tool0;
	MoveL Offs(p0,135.0,116.0, 0), v10, z5, tool0;
	MoveL Offs(p0,135.0,116.0, 0), v10, z5, tool0;
	MoveL Offs(p0,134.0,116.0, 0), v10, z5, tool0;
	MoveL Offs(p0,134.0,117.0, 0), v10, z5, tool0;
	MoveL Offs(p0,134.0,117.0, 0), v10, z5, tool0;
	MoveL Offs(p0,134.0,118.0, 0), v10, z5, tool0;
	MoveL Offs(p0,134.0,120.0, 0), v10, z5, tool0;
	MoveL Offs(p0,134.0,120.0, 0), v10, z5, tool0;
	MoveL Offs(p0,134.0,120.0, 0), v10, z5, tool0;
	MoveL Offs(p0,135.0,121.0, 0), v10, z5, tool0;
	MoveL Offs(p0,138.0,125.0, 0), v10, z5, tool0;
	MoveL Offs(p0,140.0,127.0, 0), v10, z5, tool0;
	MoveL Offs(p0,143.0,130.0, 0), v10, z5, tool0;
	MoveL Offs(p0,146.0,133.0, 0), v10, z5, tool0;
	MoveL Offs(p0,148.0,135.0, 0), v10, z5, tool0;
	MoveL Offs(p0,151.0,138.0, 0), v10, z5, tool0;
	MoveL Offs(p0,154.0,140.0, 0), v10, z5, tool0;
	MoveL Offs(p0,157.0,143.0, 0), v10, z5, tool0;
	MoveL Offs(p0,159.0,145.0, 0), v10, z5, tool0;
	MoveL Offs(p0,161.0,147.0, 0), v10, z5, tool0;
	MoveL Offs(p0,162.0,147.0, 0), v10, z5, tool0;
	MoveL Offs(p0,163.0,148.0, 0), v10, z5, tool0;
	MoveL Offs(p0,164.0,149.0, 0), v10, z5, tool0;
	MoveL Offs(p0,165.0,149.0, 0), v10, z5, tool0;
	MoveL Offs(p0,166.0,150.0, 0), v10, z5, tool0;
	MoveL Offs(p0,166.0,150.0, 0), v10, z5, tool0;
	MoveL Offs(p0,167.0,150.0, 0), v10, z5, tool0;
	MoveL Offs(p0,167.0,150.0, 0), v10, z5, tool0;
	MoveL Offs(p0,166.0,148.0, 0), v10, z5, tool0;
	MoveL Offs(p0,166.0,148.0, 0), v10, z5, tool0;
	MoveJ Offs(p0,166.0,148.0, 20), v10, z1, tool0;
	MoveJ Offs(p0,98.0,148.0, 20), v10, z1, tool0;
	MoveJ Offs(p0,98.0,148.0, 0), v10, z1, tool0;
	MoveL Offs(p0,100.0,147.0, 0), v10, z5, tool0;
	MoveL Offs(p0,101.0,147.0, 0), v10, z5, tool0;
	MoveL Offs(p0,101.0,146.0, 0), v10, z5, tool0;
	MoveL Offs(p0,102.0,146.0, 0), v10, z5, tool0;
	MoveL Offs(p0,102.0,146.0, 0), v10, z5, tool0;
	MoveL Offs(p0,103.0,146.0, 0), v10, z5, tool0;
	MoveL Offs(p0,105.0,145.0, 0), v10, z5, tool0;
	MoveL Offs(p0,101.0,145.0, 0), v10, z5, tool0;
	MoveL Offs(p0,98.0,145.0, 0), v10, z5, tool0;
	MoveL Offs(p0,98.0,145.0, 0), v10, z5, tool0;
	MoveL Offs(p0,97.0,145.0, 0), v10, z5, tool0;
	MoveL Offs(p0,96.0,145.0, 0), v10, z5, tool0;
	MoveL Offs(p0,96.0,145.0, 0), v10, z5, tool0;
	MoveL Offs(p0,95.0,145.0, 0), v10, z5, tool0;
	MoveL Offs(p0,95.0,145.0, 0), v10, z5, tool0;
	MoveL Offs(p0,94.0,145.0, 0), v10, z5, tool0;
	MoveL Offs(p0,92.0,144.0, 0), v10, z5, tool0;
	MoveL Offs(p0,91.0,146.0, 0), v10, z5, tool0;
	MoveL Offs(p0,89.0,148.0, 0), v10, z5, tool0;
	MoveL Offs(p0,89.0,148.0, 0), v10, z5, tool0;
	MoveL Offs(p0,89.0,149.0, 0), v10, z5, tool0;
	MoveL Offs(p0,90.0,149.0, 0), v10, z5, tool0;
	MoveL Offs(p0,91.0,149.0, 0), v10, z5, tool0;
	MoveL Offs(p0,91.0,149.0, 0), v10, z5, tool0;
	MoveL Offs(p0,92.0,149.0, 0), v10, z5, tool0;
	MoveL Offs(p0,95.0,148.0, 0), v10, z5, tool0;
	MoveL Offs(p0,95.0,148.0, 0), v10, z5, tool0;
	MoveL Offs(p0,96.0,148.0, 0), v10, z5, tool0;
	MoveL Offs(p0,96.0,148.0, 0), v10, z5, tool0;
	MoveL Offs(p0,97.0,148.0, 0), v10, z5, tool0;
	MoveL Offs(p0,97.0,148.0, 0), v10, z5, tool0;
	MoveL Offs(p0,98.0,148.0, 0), v10, z5, tool0;
	MoveL Offs(p0,98.0,148.0, 0), v10, z5, tool0;
	MoveJ Offs(p0,98.0,148.0, 20), v10, z1, tool0;
	MoveJ Offs(p0,115.0,145.0, 20), v10, z1, tool0;
	MoveJ Offs(p0,115.0,145.0, 0), v10, z1, tool0;
	MoveL Offs(p0,113.0,142.0, 0), v10, z5, tool0;
	MoveL Offs(p0,111.0,143.0, 0), v10, z5, tool0;
	MoveL Offs(p0,109.0,144.0, 0), v10, z5, tool0;
	MoveL Offs(p0,109.0,144.0, 0), v10, z5, tool0;
	MoveL Offs(p0,108.0,144.0, 0), v10, z5, tool0;
	MoveL Offs(p0,108.0,144.0, 0), v10, z5, tool0;
	MoveL Offs(p0,106.0,145.0, 0), v10, z5, tool0;
	MoveL Offs(p0,109.0,145.0, 0), v10, z5, tool0;
	MoveL Offs(p0,111.0,145.0, 0), v10, z5, tool0;
	MoveL Offs(p0,112.0,145.0, 0), v10, z5, tool0;
	MoveL Offs(p0,112.0,145.0, 0), v10, z5, tool0;
	MoveL Offs(p0,113.0,145.0, 0), v10, z5, tool0;
	MoveL Offs(p0,114.0,145.0, 0), v10, z5, tool0;
	MoveL Offs(p0,114.0,146.0, 0), v10, z5, tool0;
	MoveL Offs(p0,115.0,146.0, 0), v10, z5, tool0;
	MoveL Offs(p0,115.0,145.0, 0), v10, z5, tool0;
	MoveJ Offs(p0,115.0,145.0, 20), v10, z1, tool0;
	MoveJ Offs(p0,74.0,142.0, 20), v10, z1, tool0;
	MoveJ Offs(p0,74.0,142.0, 0), v10, z1, tool0;
	MoveL Offs(p0,73.0,140.0, 0), v10, z5, tool0;
	MoveL Offs(p0,73.0,140.0, 0), v10, z5, tool0;
	MoveL Offs(p0,71.0,138.0, 0), v10, z5, tool0;
	MoveL Offs(p0,71.0,136.0, 0), v10, z5, tool0;
	MoveL Offs(p0,70.0,135.0, 0), v10, z5, tool0;
	MoveL Offs(p0,70.0,133.0, 0), v10, z5, tool0;
	MoveL Offs(p0,69.0,132.0, 0), v10, z5, tool0;
	MoveL Offs(p0,69.0,130.0, 0), v10, z5, tool0;
	MoveL Offs(p0,68.0,129.0, 0), v10, z5, tool0;
	MoveL Offs(p0,68.0,127.0, 0), v10, z5, tool0;
	MoveL Offs(p0,68.0,125.0, 0), v10, z5, tool0;
	MoveL Offs(p0,67.0,122.0, 0), v10, z5, tool0;
	MoveL Offs(p0,64.0,122.0, 0), v10, z5, tool0;
	MoveL Offs(p0,61.0,122.0, 0), v10, z5, tool0;
	MoveL Offs(p0,61.0,122.0, 0), v10, z5, tool0;
	MoveL Offs(p0,61.0,122.0, 0), v10, z5, tool0;
	MoveL Offs(p0,60.0,123.0, 0), v10, z5, tool0;
	MoveL Offs(p0,60.0,123.0, 0), v10, z5, tool0;
	MoveL Offs(p0,60.0,124.0, 0), v10, z5, tool0;
	MoveL Offs(p0,60.0,125.0, 0), v10, z5, tool0;
	MoveL Offs(p0,61.0,126.0, 0), v10, z5, tool0;
	MoveL Offs(p0,61.0,128.0, 0), v10, z5, tool0;
	MoveL Offs(p0,61.0,130.0, 0), v10, z5, tool0;
	MoveL Offs(p0,62.0,133.0, 0), v10, z5, tool0;
	MoveL Offs(p0,63.0,135.0, 0), v10, z5, tool0;
	MoveL Offs(p0,64.0,136.0, 0), v10, z5, tool0;
	MoveL Offs(p0,66.0,138.0, 0), v10, z5, tool0;
	MoveL Offs(p0,67.0,140.0, 0), v10, z5, tool0;
	MoveL Offs(p0,68.0,141.0, 0), v10, z5, tool0;
	MoveL Offs(p0,70.0,143.0, 0), v10, z5, tool0;
	MoveL Offs(p0,72.0,144.0, 0), v10, z5, tool0;
	MoveL Offs(p0,74.0,144.0, 0), v10, z5, tool0;
	MoveL Offs(p0,74.0,142.0, 0), v10, z5, tool0;
	MoveJ Offs(p0,74.0,142.0, 20), v10, z1, tool0;
	MoveJ Offs(p0,108.0,143.0, 20), v10, z1, tool0;
	MoveJ Offs(p0,108.0,143.0, 0), v10, z1, tool0;
	MoveL Offs(p0,110.0,142.0, 0), v10, z5, tool0;
	MoveL Offs(p0,110.0,142.0, 0), v10, z5, tool0;
	MoveL Offs(p0,111.0,142.0, 0), v10, z5, tool0;
	MoveL Offs(p0,112.0,141.0, 0), v10, z5, tool0;
	MoveL Offs(p0,109.0,137.0, 0), v10, z5, tool0;
	MoveL Offs(p0,107.0,135.0, 0), v10, z5, tool0;
	MoveL Offs(p0,107.0,135.0, 0), v10, z5, tool0;
	MoveL Offs(p0,106.0,134.0, 0), v10, z5, tool0;
	MoveL Offs(p0,106.0,134.0, 0), v10, z5, tool0;
	MoveL Offs(p0,105.0,133.0, 0), v10, z5, tool0;
	MoveL Offs(p0,105.0,133.0, 0), v10, z5, tool0;
	MoveL Offs(p0,105.0,133.0, 0), v10, z5, tool0;
	MoveL Offs(p0,103.0,133.0, 0), v10, z5, tool0;
	MoveL Offs(p0,100.0,135.0, 0), v10, z5, tool0;
	MoveL Offs(p0,99.0,136.0, 0), v10, z5, tool0;
	MoveL Offs(p0,98.0,138.0, 0), v10, z5, tool0;
	MoveL Offs(p0,97.0,139.0, 0), v10, z5, tool0;
	MoveL Offs(p0,95.0,140.0, 0), v10, z5, tool0;
	MoveL Offs(p0,95.0,141.0, 0), v10, z5, tool0;
	MoveL Offs(p0,94.0,142.0, 0), v10, z5, tool0;
	MoveL Offs(p0,94.0,142.0, 0), v10, z5, tool0;
	MoveL Offs(p0,99.0,144.0, 0), v10, z5, tool0;
	MoveL Offs(p0,100.0,144.0, 0), v10, z5, tool0;
	MoveL Offs(p0,102.0,144.0, 0), v10, z5, tool0;
	MoveL Offs(p0,103.0,144.0, 0), v10, z5, tool0;
	MoveL Offs(p0,105.0,144.0, 0), v10, z5, tool0;
	MoveL Offs(p0,106.0,144.0, 0), v10, z5, tool0;
	MoveL Offs(p0,107.0,143.0, 0), v10, z5, tool0;
	MoveL Offs(p0,108.0,143.0, 0), v10, z5, tool0;
	MoveL Offs(p0,108.0,143.0, 0), v10, z5, tool0;
	MoveJ Offs(p0,108.0,143.0, 20), v10, z1, tool0;
	MoveJ Offs(p0,134.0,142.0, 20), v10, z1, tool0;
	MoveJ Offs(p0,134.0,142.0, 0), v10, z1, tool0;
	MoveL Offs(p0,132.0,140.0, 0), v10, z5, tool0;
	MoveL Offs(p0,131.0,139.0, 0), v10, z5, tool0;
	MoveL Offs(p0,129.0,138.0, 0), v10, z5, tool0;
	MoveL Offs(p0,128.0,138.0, 0), v10, z5, tool0;
	MoveL Offs(p0,127.0,137.0, 0), v10, z5, tool0;
	MoveL Offs(p0,126.0,137.0, 0), v10, z5, tool0;
	MoveL Offs(p0,125.0,137.0, 0), v10, z5, tool0;
	MoveL Offs(p0,124.0,137.0, 0), v10, z5, tool0;
	MoveL Offs(p0,123.0,137.0, 0), v10, z5, tool0;
	MoveL Offs(p0,123.0,136.0, 0), v10, z5, tool0;
	MoveL Offs(p0,122.0,136.0, 0), v10, z5, tool0;
	MoveL Offs(p0,123.0,140.0, 0), v10, z5, tool0;
	MoveL Offs(p0,123.0,140.0, 0), v10, z5, tool0;
	MoveL Offs(p0,124.0,141.0, 0), v10, z5, tool0;
	MoveL Offs(p0,127.0,141.0, 0), v10, z5, tool0;
	MoveL Offs(p0,127.0,142.0, 0), v10, z5, tool0;
	MoveL Offs(p0,128.0,142.0, 0), v10, z5, tool0;
	MoveL Offs(p0,129.0,142.0, 0), v10, z5, tool0;
	MoveL Offs(p0,129.0,142.0, 0), v10, z5, tool0;
	MoveL Offs(p0,130.0,143.0, 0), v10, z5, tool0;
	MoveL Offs(p0,130.0,143.0, 0), v10, z5, tool0;
	MoveL Offs(p0,132.0,143.0, 0), v10, z5, tool0;
	MoveL Offs(p0,133.0,144.0, 0), v10, z5, tool0;
	MoveL Offs(p0,133.0,143.0, 0), v10, z5, tool0;
	MoveL Offs(p0,133.0,143.0, 0), v10, z5, tool0;
	MoveL Offs(p0,133.0,143.0, 0), v10, z5, tool0;
	MoveL Offs(p0,134.0,143.0, 0), v10, z5, tool0;
	MoveL Offs(p0,134.0,142.0, 0), v10, z5, tool0;
	MoveL Offs(p0,134.0,142.0, 0), v10, z5, tool0;
	MoveL Offs(p0,134.0,142.0, 0), v10, z5, tool0;
	MoveJ Offs(p0,134.0,142.0, 20), v10, z1, tool0;
	MoveJ Offs(p0,80.0,140.0, 20), v10, z1, tool0;
	MoveJ Offs(p0,80.0,140.0, 0), v10, z1, tool0;
	MoveL Offs(p0,82.0,139.0, 0), v10, z5, tool0;
	MoveL Offs(p0,82.0,138.0, 0), v10, z5, tool0;
	MoveL Offs(p0,82.0,138.0, 0), v10, z5, tool0;
	MoveL Offs(p0,83.0,138.0, 0), v10, z5, tool0;
	MoveL Offs(p0,82.0,138.0, 0), v10, z5, tool0;
	MoveL Offs(p0,82.0,137.0, 0), v10, z5, tool0;
	MoveL Offs(p0,82.0,137.0, 0), v10, z5, tool0;
	MoveL Offs(p0,81.0,136.0, 0), v10, z5, tool0;
	MoveL Offs(p0,79.0,133.0, 0), v10, z5, tool0;
	MoveL Offs(p0,79.0,132.0, 0), v10, z5, tool0;
	MoveL Offs(p0,78.0,131.0, 0), v10, z5, tool0;
	MoveL Offs(p0,78.0,130.0, 0), v10, z5, tool0;
	MoveL Offs(p0,78.0,128.0, 0), v10, z5, tool0;
	MoveL Offs(p0,77.0,127.0, 0), v10, z5, tool0;
	MoveL Offs(p0,77.0,126.0, 0), v10, z5, tool0;
	MoveL Offs(p0,77.0,124.0, 0), v10, z5, tool0;
	MoveL Offs(p0,77.0,123.0, 0), v10, z5, tool0;
	MoveL Offs(p0,75.0,122.0, 0), v10, z5, tool0;
	MoveL Offs(p0,72.0,122.0, 0), v10, z5, tool0;
	MoveL Offs(p0,71.0,122.0, 0), v10, z5, tool0;
	MoveL Offs(p0,71.0,122.0, 0), v10, z5, tool0;
	MoveL Offs(p0,70.0,122.0, 0), v10, z5, tool0;
	MoveL Offs(p0,70.0,122.0, 0), v10, z5, tool0;
	MoveL Offs(p0,69.0,122.0, 0), v10, z5, tool0;
	MoveL Offs(p0,69.0,122.0, 0), v10, z5, tool0;
	MoveL Offs(p0,69.0,122.0, 0), v10, z5, tool0;
	MoveL Offs(p0,69.0,125.0, 0), v10, z5, tool0;
	MoveL Offs(p0,69.0,126.0, 0), v10, z5, tool0;
	MoveL Offs(p0,70.0,127.0, 0), v10, z5, tool0;
	MoveL Offs(p0,70.0,129.0, 0), v10, z5, tool0;
	MoveL Offs(p0,70.0,130.0, 0), v10, z5, tool0;
	MoveL Offs(p0,70.0,131.0, 0), v10, z5, tool0;
	MoveL Offs(p0,71.0,132.0, 0), v10, z5, tool0;
	MoveL Offs(p0,71.0,133.0, 0), v10, z5, tool0;
	MoveL Offs(p0,72.0,135.0, 0), v10, z5, tool0;
	MoveL Offs(p0,72.0,136.0, 0), v10, z5, tool0;
	MoveL Offs(p0,72.0,136.0, 0), v10, z5, tool0;
	MoveL Offs(p0,73.0,137.0, 0), v10, z5, tool0;
	MoveL Offs(p0,73.0,138.0, 0), v10, z5, tool0;
	MoveL Offs(p0,74.0,138.0, 0), v10, z5, tool0;
	MoveL Offs(p0,74.0,139.0, 0), v10, z5, tool0;
	MoveL Offs(p0,74.0,139.0, 0), v10, z5, tool0;
	MoveL Offs(p0,78.0,141.0, 0), v10, z5, tool0;
	MoveL Offs(p0,78.0,141.0, 0), v10, z5, tool0;
	MoveL Offs(p0,79.0,141.0, 0), v10, z5, tool0;
	MoveL Offs(p0,80.0,140.0, 0), v10, z5, tool0;
	MoveL Offs(p0,80.0,140.0, 0), v10, z5, tool0;
	MoveJ Offs(p0,80.0,140.0, 20), v10, z1, tool0;
	MoveJ Offs(p0,139.0,140.0, 20), v10, z1, tool0;
	MoveJ Offs(p0,139.0,140.0, 0), v10, z1, tool0;
	MoveL Offs(p0,139.0,136.0, 0), v10, z5, tool0;
	MoveL Offs(p0,138.0,135.0, 0), v10, z5, tool0;
	MoveL Offs(p0,138.0,135.0, 0), v10, z5, tool0;
	MoveL Offs(p0,137.0,134.0, 0), v10, z5, tool0;
	MoveL Offs(p0,137.0,133.0, 0), v10, z5, tool0;
	MoveL Offs(p0,135.0,130.0, 0), v10, z5, tool0;
	MoveL Offs(p0,134.0,128.0, 0), v10, z5, tool0;
	MoveL Offs(p0,133.0,127.0, 0), v10, z5, tool0;
	MoveL Offs(p0,133.0,126.0, 0), v10, z5, tool0;
	MoveL Offs(p0,132.0,125.0, 0), v10, z5, tool0;
	MoveL Offs(p0,132.0,124.0, 0), v10, z5, tool0;
	MoveL Offs(p0,131.0,123.0, 0), v10, z5, tool0;
	MoveL Offs(p0,131.0,123.0, 0), v10, z5, tool0;
	MoveL Offs(p0,131.0,122.0, 0), v10, z5, tool0;
	MoveL Offs(p0,132.0,120.0, 0), v10, z5, tool0;
	MoveL Offs(p0,132.0,119.0, 0), v10, z5, tool0;
	MoveL Offs(p0,132.0,118.0, 0), v10, z5, tool0;
	MoveL Offs(p0,132.0,117.0, 0), v10, z5, tool0;
	MoveL Offs(p0,133.0,116.0, 0), v10, z5, tool0;
	MoveL Offs(p0,133.0,116.0, 0), v10, z5, tool0;
	MoveL Offs(p0,133.0,115.0, 0), v10, z5, tool0;
	MoveL Offs(p0,133.0,115.0, 0), v10, z5, tool0;
	MoveL Offs(p0,135.0,114.0, 0), v10, z5, tool0;
	MoveL Offs(p0,136.0,114.0, 0), v10, z5, tool0;
	MoveL Offs(p0,136.0,114.0, 0), v10, z5, tool0;
	MoveL Offs(p0,138.0,114.0, 0), v10, z5, tool0;
	MoveL Offs(p0,138.0,114.0, 0), v10, z5, tool0;
	MoveL Offs(p0,138.0,113.0, 0), v10, z5, tool0;
	MoveL Offs(p0,139.0,113.0, 0), v10, z5, tool0;
	MoveL Offs(p0,139.0,113.0, 0), v10, z5, tool0;
	MoveL Offs(p0,139.0,111.0, 0), v10, z5, tool0;
	MoveL Offs(p0,139.0,110.0, 0), v10, z5, tool0;
	MoveL Offs(p0,138.0,110.0, 0), v10, z5, tool0;
	MoveL Offs(p0,138.0,109.0, 0), v10, z5, tool0;
	MoveL Offs(p0,138.0,109.0, 0), v10, z5, tool0;
	MoveL Offs(p0,136.0,105.0, 0), v10, z5, tool0;
	MoveL Offs(p0,135.0,105.0, 0), v10, z5, tool0;
	MoveL Offs(p0,135.0,104.0, 0), v10, z5, tool0;
	MoveL Offs(p0,135.0,104.0, 0), v10, z5, tool0;
	MoveL Offs(p0,135.0,104.0, 0), v10, z5, tool0;
	MoveL Offs(p0,134.0,101.0, 0), v10, z5, tool0;
	MoveL Offs(p0,134.0,101.0, 0), v10, z5, tool0;
	MoveL Offs(p0,134.0,100.0, 0), v10, z5, tool0;
	MoveL Offs(p0,134.0,100.0, 0), v10, z5, tool0;
	MoveL Offs(p0,134.0,99.0, 0), v10, z5, tool0;
	MoveL Offs(p0,133.0,96.0, 0), v10, z5, tool0;
	MoveL Offs(p0,131.0,101.0, 0), v10, z5, tool0;
	MoveL Offs(p0,130.0,103.0, 0), v10, z5, tool0;
	MoveL Offs(p0,129.0,105.0, 0), v10, z5, tool0;
	MoveL Offs(p0,128.0,107.0, 0), v10, z5, tool0;
	MoveL Offs(p0,127.0,108.0, 0), v10, z5, tool0;
	MoveL Offs(p0,126.0,110.0, 0), v10, z5, tool0;
	MoveL Offs(p0,125.0,111.0, 0), v10, z5, tool0;
	MoveL Offs(p0,125.0,112.0, 0), v10, z5, tool0;
	MoveL Offs(p0,124.0,113.0, 0), v10, z5, tool0;
	MoveL Offs(p0,124.0,114.0, 0), v10, z5, tool0;
	MoveL Offs(p0,123.0,114.0, 0), v10, z5, tool0;
	MoveL Offs(p0,121.0,115.0, 0), v10, z5, tool0;
	MoveL Offs(p0,120.0,115.0, 0), v10, z5, tool0;
	MoveL Offs(p0,120.0,115.0, 0), v10, z5, tool0;
	MoveL Offs(p0,119.0,115.0, 0), v10, z5, tool0;
	MoveL Offs(p0,119.0,115.0, 0), v10, z5, tool0;
	MoveL Offs(p0,118.0,114.0, 0), v10, z5, tool0;
	MoveL Offs(p0,118.0,114.0, 0), v10, z5, tool0;
	MoveL Offs(p0,116.0,114.0, 0), v10, z5, tool0;
	MoveL Offs(p0,115.0,114.0, 0), v10, z5, tool0;
	MoveL Offs(p0,115.0,114.0, 0), v10, z5, tool0;
	MoveL Offs(p0,115.0,114.0, 0), v10, z5, tool0;
	MoveL Offs(p0,114.0,114.0, 0), v10, z5, tool0;
	MoveL Offs(p0,117.0,117.0, 0), v10, z5, tool0;
	MoveL Offs(p0,118.0,119.0, 0), v10, z5, tool0;
	MoveL Offs(p0,118.0,120.0, 0), v10, z5, tool0;
	MoveL Offs(p0,118.0,121.0, 0), v10, z5, tool0;
	MoveL Offs(p0,118.0,122.0, 0), v10, z5, tool0;
	MoveL Offs(p0,118.0,124.0, 0), v10, z5, tool0;
	MoveL Offs(p0,117.0,125.0, 0), v10, z5, tool0;
	MoveL Offs(p0,116.0,126.0, 0), v10, z5, tool0;
	MoveL Offs(p0,115.0,129.0, 0), v10, z5, tool0;
	MoveL Offs(p0,117.0,132.0, 0), v10, z5, tool0;
	MoveL Offs(p0,118.0,134.0, 0), v10, z5, tool0;
	MoveL Offs(p0,118.0,134.0, 0), v10, z5, tool0;
	MoveL Offs(p0,119.0,135.0, 0), v10, z5, tool0;
	MoveL Offs(p0,119.0,135.0, 0), v10, z5, tool0;
	MoveL Offs(p0,119.0,135.0, 0), v10, z5, tool0;
	MoveL Offs(p0,120.0,135.0, 0), v10, z5, tool0;
	MoveL Offs(p0,120.0,135.0, 0), v10, z5, tool0;
	MoveL Offs(p0,120.0,135.0, 0), v10, z5, tool0;
	MoveL Offs(p0,121.0,135.0, 0), v10, z5, tool0;
	MoveL Offs(p0,123.0,135.0, 0), v10, z5, tool0;
	MoveL Offs(p0,123.0,135.0, 0), v10, z5, tool0;
	MoveL Offs(p0,124.0,135.0, 0), v10, z5, tool0;
	MoveL Offs(p0,124.0,135.0, 0), v10, z5, tool0;
	MoveL Offs(p0,127.0,136.0, 0), v10, z5, tool0;
	MoveL Offs(p0,128.0,137.0, 0), v10, z5, tool0;
	MoveL Offs(p0,130.0,137.0, 0), v10, z5, tool0;
	MoveL Offs(p0,131.0,138.0, 0), v10, z5, tool0;
	MoveL Offs(p0,133.0,139.0, 0), v10, z5, tool0;
	MoveL Offs(p0,134.0,139.0, 0), v10, z5, tool0;
	MoveL Offs(p0,136.0,140.0, 0), v10, z5, tool0;
	MoveL Offs(p0,137.0,140.0, 0), v10, z5, tool0;
	MoveL Offs(p0,139.0,141.0, 0), v10, z5, tool0;
	MoveL Offs(p0,139.0,141.0, 0), v10, z5, tool0;
	MoveL Offs(p0,139.0,141.0, 0), v10, z5, tool0;
	MoveL Offs(p0,139.0,140.0, 0), v10, z5, tool0;
	MoveL Offs(p0,139.0,140.0, 0), v10, z5, tool0;
	MoveJ Offs(p0,139.0,140.0, 20), v10, z1, tool0;
	MoveJ Offs(p0,87.0,131.0, 20), v10, z1, tool0;
	MoveJ Offs(p0,87.0,131.0, 0), v10, z1, tool0;
	MoveL Offs(p0,88.0,129.0, 0), v10, z5, tool0;
	MoveL Offs(p0,88.0,128.0, 0), v10, z5, tool0;
	MoveL Offs(p0,89.0,128.0, 0), v10, z5, tool0;
	MoveL Offs(p0,89.0,127.0, 0), v10, z5, tool0;
	MoveL Offs(p0,89.0,127.0, 0), v10, z5, tool0;
	MoveL Offs(p0,89.0,126.0, 0), v10, z5, tool0;
	MoveL Offs(p0,89.0,126.0, 0), v10, z5, tool0;
	MoveL Offs(p0,89.0,125.0, 0), v10, z5, tool0;
	MoveL Offs(p0,90.0,124.0, 0), v10, z5, tool0;
	MoveL Offs(p0,87.0,124.0, 0), v10, z5, tool0;
	MoveL Offs(p0,84.0,123.0, 0), v10, z5, tool0;
	MoveL Offs(p0,84.0,123.0, 0), v10, z5, tool0;
	MoveL Offs(p0,83.0,123.0, 0), v10, z5, tool0;
	MoveL Offs(p0,83.0,123.0, 0), v10, z5, tool0;
	MoveL Offs(p0,82.0,123.0, 0), v10, z5, tool0;
	MoveL Offs(p0,82.0,123.0, 0), v10, z5, tool0;
	MoveL Offs(p0,81.0,123.0, 0), v10, z5, tool0;
	MoveL Offs(p0,79.0,123.0, 0), v10, z5, tool0;
	MoveL Offs(p0,79.0,125.0, 0), v10, z5, tool0;
	MoveL Offs(p0,79.0,128.0, 0), v10, z5, tool0;
	MoveL Offs(p0,79.0,129.0, 0), v10, z5, tool0;
	MoveL Offs(p0,80.0,130.0, 0), v10, z5, tool0;
	MoveL Offs(p0,80.0,131.0, 0), v10, z5, tool0;
	MoveL Offs(p0,80.0,132.0, 0), v10, z5, tool0;
	MoveL Offs(p0,81.0,133.0, 0), v10, z5, tool0;
	MoveL Offs(p0,82.0,134.0, 0), v10, z5, tool0;
	MoveL Offs(p0,82.0,135.0, 0), v10, z5, tool0;
	MoveL Offs(p0,83.0,136.0, 0), v10, z5, tool0;
	MoveL Offs(p0,85.0,136.0, 0), v10, z5, tool0;
	MoveL Offs(p0,86.0,135.0, 0), v10, z5, tool0;
	MoveL Offs(p0,86.0,133.0, 0), v10, z5, tool0;
	MoveL Offs(p0,87.0,131.0, 0), v10, z5, tool0;
	MoveL Offs(p0,87.0,131.0, 0), v10, z5, tool0;
	MoveJ Offs(p0,87.0,131.0, 20), v10, z1, tool0;
	MoveJ Offs(p0,116.0,125.0, 20), v10, z1, tool0;
	MoveJ Offs(p0,116.0,125.0, 0), v10, z1, tool0;
	MoveL Offs(p0,117.0,122.0, 0), v10, z5, tool0;
	MoveL Offs(p0,117.0,121.0, 0), v10, z5, tool0;
	MoveL Offs(p0,117.0,120.0, 0), v10, z5, tool0;
	MoveL Offs(p0,117.0,119.0, 0), v10, z5, tool0;
	MoveL Offs(p0,117.0,119.0, 0), v10, z5, tool0;
	MoveL Offs(p0,117.0,118.0, 0), v10, z5, tool0;
	MoveL Offs(p0,116.0,117.0, 0), v10, z5, tool0;
	MoveL Offs(p0,116.0,117.0, 0), v10, z5, tool0;
	MoveL Offs(p0,113.0,118.0, 0), v10, z5, tool0;
	MoveL Offs(p0,113.0,119.0, 0), v10, z5, tool0;
	MoveL Offs(p0,113.0,119.0, 0), v10, z5, tool0;
	MoveL Offs(p0,111.0,121.0, 0), v10, z5, tool0;
	MoveL Offs(p0,113.0,124.0, 0), v10, z5, tool0;
	MoveL Offs(p0,114.0,126.0, 0), v10, z5, tool0;
	MoveL Offs(p0,114.0,126.0, 0), v10, z5, tool0;
	MoveL Offs(p0,114.0,127.0, 0), v10, z5, tool0;
	MoveL Offs(p0,114.0,127.0, 0), v10, z5, tool0;
	MoveL Offs(p0,115.0,127.0, 0), v10, z5, tool0;
	MoveL Offs(p0,116.0,125.0, 0), v10, z5, tool0;
	MoveJ Offs(p0,116.0,125.0, 20), v10, z1, tool0;
	MoveJ Offs(p0,20.0,121.0, 20), v10, z1, tool0;
	MoveJ Offs(p0,20.0,121.0, 0), v10, z1, tool0;
	MoveL Offs(p0,25.0,116.0, 0), v10, z5, tool0;
	MoveL Offs(p0,25.0,115.0, 0), v10, z5, tool0;
	MoveL Offs(p0,25.0,114.0, 0), v10, z5, tool0;
	MoveL Offs(p0,25.0,113.0, 0), v10, z5, tool0;
	MoveL Offs(p0,25.0,111.0, 0), v10, z5, tool0;
	MoveL Offs(p0,25.0,110.0, 0), v10, z5, tool0;
	MoveL Offs(p0,25.0,108.0, 0), v10, z5, tool0;
	MoveL Offs(p0,25.0,106.0, 0), v10, z5, tool0;
	MoveL Offs(p0,25.0,104.0, 0), v10, z5, tool0;
	MoveL Offs(p0,25.0,102.0, 0), v10, z5, tool0;
	MoveL Offs(p0,25.0,100.0, 0), v10, z5, tool0;
	MoveL Offs(p0,25.0,99.0, 0), v10, z5, tool0;
	MoveL Offs(p0,25.0,98.0, 0), v10, z5, tool0;
	MoveL Offs(p0,25.0,96.0, 0), v10, z5, tool0;
	MoveL Offs(p0,24.0,95.0, 0), v10, z5, tool0;
	MoveL Offs(p0,24.0,94.0, 0), v10, z5, tool0;
	MoveL Offs(p0,24.0,93.0, 0), v10, z5, tool0;
	MoveL Offs(p0,23.0,92.0, 0), v10, z5, tool0;
	MoveL Offs(p0,23.0,90.0, 0), v10, z5, tool0;
	MoveL Offs(p0,21.0,91.0, 0), v10, z5, tool0;
	MoveL Offs(p0,19.0,94.0, 0), v10, z5, tool0;
	MoveL Offs(p0,19.0,95.0, 0), v10, z5, tool0;
	MoveL Offs(p0,19.0,96.0, 0), v10, z5, tool0;
	MoveL Offs(p0,19.0,98.0, 0), v10, z5, tool0;
	MoveL Offs(p0,20.0,102.0, 0), v10, z5, tool0;
	MoveL Offs(p0,20.0,104.0, 0), v10, z5, tool0;
	MoveL Offs(p0,20.0,107.0, 0), v10, z5, tool0;
	MoveL Offs(p0,20.0,109.0, 0), v10, z5, tool0;
	MoveL Offs(p0,20.0,111.0, 0), v10, z5, tool0;
	MoveL Offs(p0,20.0,113.0, 0), v10, z5, tool0;
	MoveL Offs(p0,19.0,115.0, 0), v10, z5, tool0;
	MoveL Offs(p0,19.0,116.0, 0), v10, z5, tool0;
	MoveL Offs(p0,18.0,118.0, 0), v10, z5, tool0;
	MoveL Offs(p0,19.0,123.0, 0), v10, z5, tool0;
	MoveL Offs(p0,19.0,123.0, 0), v10, z5, tool0;
	MoveL Offs(p0,19.0,123.0, 0), v10, z5, tool0;
	MoveL Offs(p0,19.0,123.0, 0), v10, z5, tool0;
	MoveL Offs(p0,19.0,123.0, 0), v10, z5, tool0;
	MoveL Offs(p0,19.0,123.0, 0), v10, z5, tool0;
	MoveL Offs(p0,19.0,123.0, 0), v10, z5, tool0;
	MoveL Offs(p0,20.0,121.0, 0), v10, z5, tool0;
	MoveJ Offs(p0,20.0,121.0, 20), v10, z1, tool0;
	MoveJ Offs(p0,158.0,121.0, 20), v10, z1, tool0;
	MoveJ Offs(p0,158.0,121.0, 0), v10, z1, tool0;
	MoveL Offs(p0,156.0,118.0, 0), v10, z5, tool0;
	MoveL Offs(p0,156.0,118.0, 0), v10, z5, tool0;
	MoveL Offs(p0,155.0,117.0, 0), v10, z5, tool0;
	MoveL Offs(p0,155.0,116.0, 0), v10, z5, tool0;
	MoveL Offs(p0,155.0,116.0, 0), v10, z5, tool0;
	MoveL Offs(p0,155.0,115.0, 0), v10, z5, tool0;
	MoveL Offs(p0,155.0,114.0, 0), v10, z5, tool0;
	MoveL Offs(p0,155.0,112.0, 0), v10, z5, tool0;
	MoveL Offs(p0,155.0,112.0, 0), v10, z5, tool0;
	MoveL Offs(p0,156.0,111.0, 0), v10, z5, tool0;
	MoveL Offs(p0,156.0,111.0, 0), v10, z5, tool0;
	MoveL Offs(p0,156.0,110.0, 0), v10, z5, tool0;
	MoveL Offs(p0,157.0,110.0, 0), v10, z5, tool0;
	MoveL Offs(p0,157.0,109.0, 0), v10, z5, tool0;
	MoveL Offs(p0,159.0,107.0, 0), v10, z5, tool0;
	MoveL Offs(p0,159.0,107.0, 0), v10, z5, tool0;
	MoveL Offs(p0,159.0,106.0, 0), v10, z5, tool0;
	MoveL Offs(p0,159.0,106.0, 0), v10, z5, tool0;
	MoveL Offs(p0,158.0,106.0, 0), v10, z5, tool0;
	MoveL Offs(p0,158.0,105.0, 0), v10, z5, tool0;
	MoveL Offs(p0,156.0,104.0, 0), v10, z5, tool0;
	MoveL Offs(p0,155.0,104.0, 0), v10, z5, tool0;
	MoveL Offs(p0,153.0,104.0, 0), v10, z5, tool0;
	MoveL Offs(p0,152.0,104.0, 0), v10, z5, tool0;
	MoveL Offs(p0,150.0,104.0, 0), v10, z5, tool0;
	MoveL Offs(p0,146.0,104.0, 0), v10, z5, tool0;
	MoveL Offs(p0,145.0,104.0, 0), v10, z5, tool0;
	MoveL Offs(p0,144.0,104.0, 0), v10, z5, tool0;
	MoveL Offs(p0,143.0,104.0, 0), v10, z5, tool0;
	MoveL Offs(p0,142.0,104.0, 0), v10, z5, tool0;
	MoveL Offs(p0,141.0,104.0, 0), v10, z5, tool0;
	MoveL Offs(p0,140.0,104.0, 0), v10, z5, tool0;
	MoveL Offs(p0,140.0,104.0, 0), v10, z5, tool0;
	MoveL Offs(p0,139.0,103.0, 0), v10, z5, tool0;
	MoveL Offs(p0,137.0,103.0, 0), v10, z5, tool0;
	MoveL Offs(p0,137.0,103.0, 0), v10, z5, tool0;
	MoveL Offs(p0,137.0,103.0, 0), v10, z5, tool0;
	MoveL Offs(p0,136.0,103.0, 0), v10, z5, tool0;
	MoveL Offs(p0,136.0,103.0, 0), v10, z5, tool0;
	MoveL Offs(p0,138.0,105.0, 0), v10, z5, tool0;
	MoveL Offs(p0,138.0,106.0, 0), v10, z5, tool0;
	MoveL Offs(p0,138.0,106.0, 0), v10, z5, tool0;
	MoveL Offs(p0,138.0,107.0, 0), v10, z5, tool0;
	MoveL Offs(p0,140.0,109.0, 0), v10, z5, tool0;
	MoveL Offs(p0,140.0,109.0, 0), v10, z5, tool0;
	MoveL Offs(p0,140.0,110.0, 0), v10, z5, tool0;
	MoveL Offs(p0,140.0,110.0, 0), v10, z5, tool0;
	MoveL Offs(p0,140.0,111.0, 0), v10, z5, tool0;
	MoveL Offs(p0,140.0,111.0, 0), v10, z5, tool0;
	MoveL Offs(p0,140.0,111.0, 0), v10, z5, tool0;
	MoveL Offs(p0,140.0,112.0, 0), v10, z5, tool0;
	MoveL Offs(p0,141.0,114.0, 0), v10, z5, tool0;
	MoveL Offs(p0,142.0,114.0, 0), v10, z5, tool0;
	MoveL Offs(p0,145.0,116.0, 0), v10, z5, tool0;
	MoveL Offs(p0,146.0,117.0, 0), v10, z5, tool0;
	MoveL Offs(p0,147.0,117.0, 0), v10, z5, tool0;
	MoveL Offs(p0,149.0,118.0, 0), v10, z5, tool0;
	MoveL Offs(p0,150.0,119.0, 0), v10, z5, tool0;
	MoveL Offs(p0,152.0,119.0, 0), v10, z5, tool0;
	MoveL Offs(p0,153.0,120.0, 0), v10, z5, tool0;
	MoveL Offs(p0,154.0,121.0, 0), v10, z5, tool0;
	MoveL Offs(p0,156.0,121.0, 0), v10, z5, tool0;
	MoveL Offs(p0,157.0,122.0, 0), v10, z5, tool0;
	MoveL Offs(p0,158.0,122.0, 0), v10, z5, tool0;
	MoveL Offs(p0,158.0,122.0, 0), v10, z5, tool0;
	MoveL Offs(p0,158.0,122.0, 0), v10, z5, tool0;
	MoveL Offs(p0,158.0,122.0, 0), v10, z5, tool0;
	MoveL Offs(p0,158.0,121.0, 0), v10, z5, tool0;
	MoveL Offs(p0,158.0,121.0, 0), v10, z5, tool0;
	MoveL Offs(p0,158.0,121.0, 0), v10, z5, tool0;
	MoveL Offs(p0,158.0,121.0, 0), v10, z5, tool0;
	MoveJ Offs(p0,158.0,121.0, 20), v10, z1, tool0;
	MoveJ Offs(p0,10.0,106.0, 20), v10, z1, tool0;
	MoveJ Offs(p0,10.0,106.0, 0), v10, z1, tool0;
	MoveL Offs(p0,11.0,104.0, 0), v10, z5, tool0;
	MoveL Offs(p0,12.0,102.0, 0), v10, z5, tool0;
	MoveL Offs(p0,13.0,101.0, 0), v10, z5, tool0;
	MoveL Offs(p0,13.0,100.0, 0), v10, z5, tool0;
	MoveL Offs(p0,14.0,99.0, 0), v10, z5, tool0;
	MoveL Offs(p0,15.0,98.0, 0), v10, z5, tool0;
	MoveL Offs(p0,15.0,97.0, 0), v10, z5, tool0;
	MoveL Offs(p0,16.0,97.0, 0), v10, z5, tool0;
	MoveL Offs(p0,17.0,96.0, 0), v10, z5, tool0;
	MoveL Offs(p0,18.0,94.0, 0), v10, z5, tool0;
	MoveL Offs(p0,18.0,93.0, 0), v10, z5, tool0;
	MoveL Offs(p0,18.0,93.0, 0), v10, z5, tool0;
	MoveL Offs(p0,18.0,93.0, 0), v10, z5, tool0;
	MoveL Offs(p0,18.0,93.0, 0), v10, z5, tool0;
	MoveL Offs(p0,17.0,93.0, 0), v10, z5, tool0;
	MoveL Offs(p0,15.0,94.0, 0), v10, z5, tool0;
	MoveL Offs(p0,15.0,94.0, 0), v10, z5, tool0;
	MoveL Offs(p0,15.0,94.0, 0), v10, z5, tool0;
	MoveL Offs(p0,14.0,96.0, 0), v10, z5, tool0;
	MoveL Offs(p0,14.0,97.0, 0), v10, z5, tool0;
	MoveL Offs(p0,12.0,100.0, 0), v10, z5, tool0;
	MoveL Offs(p0,11.0,101.0, 0), v10, z5, tool0;
	MoveL Offs(p0,10.0,103.0, 0), v10, z5, tool0;
	MoveL Offs(p0,9.0,104.0, 0), v10, z5, tool0;
	MoveL Offs(p0,9.0,106.0, 0), v10, z5, tool0;
	MoveL Offs(p0,8.0,108.0, 0), v10, z5, tool0;
	MoveL Offs(p0,8.0,109.0, 0), v10, z5, tool0;
	MoveL Offs(p0,7.0,111.0, 0), v10, z5, tool0;
	MoveL Offs(p0,7.0,113.0, 0), v10, z5, tool0;
	MoveL Offs(p0,7.0,115.0, 0), v10, z5, tool0;
	MoveL Offs(p0,6.0,116.0, 0), v10, z5, tool0;
	MoveL Offs(p0,6.0,116.0, 0), v10, z5, tool0;
	MoveL Offs(p0,6.0,117.0, 0), v10, z5, tool0;
	MoveL Offs(p0,7.0,117.0, 0), v10, z5, tool0;
	MoveL Offs(p0,7.0,116.0, 0), v10, z5, tool0;
	MoveL Offs(p0,7.0,116.0, 0), v10, z5, tool0;
	MoveL Offs(p0,8.0,111.0, 0), v10, z5, tool0;
	MoveL Offs(p0,9.0,110.0, 0), v10, z5, tool0;
	MoveL Offs(p0,9.0,109.0, 0), v10, z5, tool0;
	MoveL Offs(p0,9.0,109.0, 0), v10, z5, tool0;
	MoveL Offs(p0,9.0,108.0, 0), v10, z5, tool0;
	MoveL Offs(p0,10.0,107.0, 0), v10, z5, tool0;
	MoveL Offs(p0,10.0,106.0, 0), v10, z5, tool0;
	MoveL Offs(p0,10.0,106.0, 0), v10, z5, tool0;
	MoveL Offs(p0,10.0,106.0, 0), v10, z5, tool0;
	MoveJ Offs(p0,10.0,106.0, 20), v10, z1, tool0;
	MoveJ Offs(p0,15.0,116.0, 20), v10, z1, tool0;
	MoveJ Offs(p0,15.0,116.0, 0), v10, z1, tool0;
	MoveL Offs(p0,15.0,117.0, 0), v10, z5, tool0;
	MoveL Offs(p0,16.0,115.0, 0), v10, z5, tool0;
	MoveL Offs(p0,17.0,114.0, 0), v10, z5, tool0;
	MoveL Offs(p0,18.0,115.0, 0), v10, z5, tool0;
	MoveL Offs(p0,19.0,112.0, 0), v10, z5, tool0;
	MoveL Offs(p0,19.0,110.0, 0), v10, z5, tool0;
	MoveL Offs(p0,19.0,108.0, 0), v10, z5, tool0;
	MoveL Offs(p0,19.0,106.0, 0), v10, z5, tool0;
	MoveL Offs(p0,19.0,104.0, 0), v10, z5, tool0;
	MoveL Offs(p0,19.0,103.0, 0), v10, z5, tool0;
	MoveL Offs(p0,19.0,101.0, 0), v10, z5, tool0;
	MoveL Offs(p0,19.0,100.0, 0), v10, z5, tool0;
	MoveL Offs(p0,18.0,98.0, 0), v10, z5, tool0;
	MoveL Offs(p0,18.0,97.0, 0), v10, z5, tool0;
	MoveL Offs(p0,18.0,97.0, 0), v10, z5, tool0;
	MoveL Offs(p0,18.0,97.0, 0), v10, z5, tool0;
	MoveL Offs(p0,18.0,96.0, 0), v10, z5, tool0;
	MoveL Offs(p0,18.0,96.0, 0), v10, z5, tool0;
	MoveL Offs(p0,17.0,96.0, 0), v10, z5, tool0;
	MoveL Offs(p0,17.0,97.0, 0), v10, z5, tool0;
	MoveL Offs(p0,17.0,97.0, 0), v10, z5, tool0;
	MoveL Offs(p0,15.0,99.0, 0), v10, z5, tool0;
	MoveL Offs(p0,14.0,101.0, 0), v10, z5, tool0;
	MoveL Offs(p0,13.0,103.0, 0), v10, z5, tool0;
	MoveL Offs(p0,12.0,105.0, 0), v10, z5, tool0;
	MoveL Offs(p0,11.0,107.0, 0), v10, z5, tool0;
	MoveL Offs(p0,10.0,109.0, 0), v10, z5, tool0;
	MoveL Offs(p0,9.0,111.0, 0), v10, z5, tool0;
	MoveL Offs(p0,8.0,113.0, 0), v10, z5, tool0;
	MoveL Offs(p0,8.0,114.0, 0), v10, z5, tool0;
	MoveL Offs(p0,10.0,114.0, 0), v10, z5, tool0;
	MoveL Offs(p0,11.0,115.0, 0), v10, z5, tool0;
	MoveL Offs(p0,12.0,117.0, 0), v10, z5, tool0;
	MoveL Offs(p0,13.0,116.0, 0), v10, z5, tool0;
	MoveL Offs(p0,14.0,114.0, 0), v10, z5, tool0;
	MoveL Offs(p0,15.0,116.0, 0), v10, z5, tool0;
	MoveL Offs(p0,15.0,116.0, 0), v10, z5, tool0;
	MoveJ Offs(p0,15.0,116.0, 20), v10, z1, tool0;
	MoveJ Offs(p0,35.0,113.0, 20), v10, z1, tool0;
	MoveJ Offs(p0,35.0,113.0, 0), v10, z1, tool0;
	MoveL Offs(p0,34.0,111.0, 0), v10, z5, tool0;
	MoveL Offs(p0,34.0,109.0, 0), v10, z5, tool0;
	MoveL Offs(p0,34.0,107.0, 0), v10, z5, tool0;
	MoveL Offs(p0,33.0,104.0, 0), v10, z5, tool0;
	MoveL Offs(p0,32.0,102.0, 0), v10, z5, tool0;
	MoveL Offs(p0,32.0,100.0, 0), v10, z5, tool0;
	MoveL Offs(p0,31.0,98.0, 0), v10, z5, tool0;
	MoveL Offs(p0,30.0,96.0, 0), v10, z5, tool0;
	MoveL Offs(p0,29.0,95.0, 0), v10, z5, tool0;
	MoveL Offs(p0,28.0,93.0, 0), v10, z5, tool0;
	MoveL Offs(p0,26.0,91.0, 0), v10, z5, tool0;
	MoveL Offs(p0,26.0,91.0, 0), v10, z5, tool0;
	MoveL Offs(p0,26.0,90.0, 0), v10, z5, tool0;
	MoveL Offs(p0,26.0,90.0, 0), v10, z5, tool0;
	MoveL Offs(p0,26.0,90.0, 0), v10, z5, tool0;
	MoveL Offs(p0,26.0,90.0, 0), v10, z5, tool0;
	MoveL Offs(p0,26.0,94.0, 0), v10, z5, tool0;
	MoveL Offs(p0,26.0,94.0, 0), v10, z5, tool0;
	MoveL Offs(p0,26.0,94.0, 0), v10, z5, tool0;
	MoveL Offs(p0,26.0,95.0, 0), v10, z5, tool0;
	MoveL Offs(p0,27.0,95.0, 0), v10, z5, tool0;
	MoveL Offs(p0,29.0,97.0, 0), v10, z5, tool0;
	MoveL Offs(p0,29.0,99.0, 0), v10, z5, tool0;
	MoveL Offs(p0,30.0,101.0, 0), v10, z5, tool0;
	MoveL Offs(p0,31.0,102.0, 0), v10, z5, tool0;
	MoveL Offs(p0,32.0,104.0, 0), v10, z5, tool0;
	MoveL Offs(p0,33.0,106.0, 0), v10, z5, tool0;
	MoveL Offs(p0,33.0,108.0, 0), v10, z5, tool0;
	MoveL Offs(p0,34.0,110.0, 0), v10, z5, tool0;
	MoveL Offs(p0,34.0,111.0, 0), v10, z5, tool0;
	MoveL Offs(p0,34.0,114.0, 0), v10, z5, tool0;
	MoveL Offs(p0,34.0,114.0, 0), v10, z5, tool0;
	MoveL Offs(p0,34.0,114.0, 0), v10, z5, tool0;
	MoveL Offs(p0,34.0,114.0, 0), v10, z5, tool0;
	MoveL Offs(p0,34.0,114.0, 0), v10, z5, tool0;
	MoveL Offs(p0,35.0,115.0, 0), v10, z5, tool0;
	MoveL Offs(p0,35.0,114.0, 0), v10, z5, tool0;
	MoveL Offs(p0,35.0,114.0, 0), v10, z5, tool0;
	MoveL Offs(p0,35.0,113.0, 0), v10, z5, tool0;
	MoveL Offs(p0,35.0,113.0, 0), v10, z5, tool0;
	MoveJ Offs(p0,35.0,113.0, 20), v10, z1, tool0;
	MoveJ Offs(p0,60.0,114.0, 20), v10, z1, tool0;
	MoveJ Offs(p0,60.0,114.0, 0), v10, z1, tool0;
	MoveL Offs(p0,60.0,112.0, 0), v10, z5, tool0;
	MoveL Offs(p0,60.0,112.0, 0), v10, z5, tool0;
	MoveL Offs(p0,60.0,112.0, 0), v10, z5, tool0;
	MoveL Offs(p0,60.0,111.0, 0), v10, z5, tool0;
	MoveL Offs(p0,59.0,109.0, 0), v10, z5, tool0;
	MoveL Offs(p0,59.0,107.0, 0), v10, z5, tool0;
	MoveL Offs(p0,59.0,105.0, 0), v10, z5, tool0;
	MoveL Offs(p0,59.0,103.0, 0), v10, z5, tool0;
	MoveL Offs(p0,59.0,101.0, 0), v10, z5, tool0;
	MoveL Offs(p0,59.0,99.0, 0), v10, z5, tool0;
	MoveL Offs(p0,60.0,97.0, 0), v10, z5, tool0;
	MoveL Offs(p0,60.0,95.0, 0), v10, z5, tool0;
	MoveL Offs(p0,61.0,94.0, 0), v10, z5, tool0;
	MoveL Offs(p0,59.0,92.0, 0), v10, z5, tool0;
	MoveL Offs(p0,59.0,92.0, 0), v10, z5, tool0;
	MoveL Offs(p0,58.0,92.0, 0), v10, z5, tool0;
	MoveL Offs(p0,58.0,92.0, 0), v10, z5, tool0;
	MoveL Offs(p0,57.0,92.0, 0), v10, z5, tool0;
	MoveL Offs(p0,57.0,92.0, 0), v10, z5, tool0;
	MoveL Offs(p0,56.0,94.0, 0), v10, z5, tool0;
	MoveL Offs(p0,56.0,95.0, 0), v10, z5, tool0;
	MoveL Offs(p0,56.0,95.0, 0), v10, z5, tool0;
	MoveL Offs(p0,56.0,96.0, 0), v10, z5, tool0;
	MoveL Offs(p0,55.0,100.0, 0), v10, z5, tool0;
	MoveL Offs(p0,55.0,102.0, 0), v10, z5, tool0;
	MoveL Offs(p0,55.0,104.0, 0), v10, z5, tool0;
	MoveL Offs(p0,55.0,106.0, 0), v10, z5, tool0;
	MoveL Offs(p0,56.0,108.0, 0), v10, z5, tool0;
	MoveL Offs(p0,56.0,110.0, 0), v10, z5, tool0;
	MoveL Offs(p0,56.0,112.0, 0), v10, z5, tool0;
	MoveL Offs(p0,57.0,114.0, 0), v10, z5, tool0;
	MoveL Offs(p0,57.0,115.0, 0), v10, z5, tool0;
	MoveL Offs(p0,60.0,115.0, 0), v10, z5, tool0;
	MoveL Offs(p0,60.0,115.0, 0), v10, z5, tool0;
	MoveL Offs(p0,60.0,114.0, 0), v10, z5, tool0;
	MoveL Offs(p0,60.0,114.0, 0), v10, z5, tool0;
	MoveJ Offs(p0,60.0,114.0, 20), v10, z1, tool0;
	MoveJ Offs(p0,63.0,114.0, 20), v10, z1, tool0;
	MoveJ Offs(p0,63.0,114.0, 0), v10, z1, tool0;
	MoveL Offs(p0,63.0,112.0, 0), v10, z5, tool0;
	MoveL Offs(p0,63.0,112.0, 0), v10, z5, tool0;
	MoveL Offs(p0,63.0,112.0, 0), v10, z5, tool0;
	MoveL Offs(p0,64.0,111.0, 0), v10, z5, tool0;
	MoveL Offs(p0,64.0,110.0, 0), v10, z5, tool0;
	MoveL Offs(p0,65.0,110.0, 0), v10, z5, tool0;
	MoveL Offs(p0,66.0,108.0, 0), v10, z5, tool0;
	MoveL Offs(p0,66.0,108.0, 0), v10, z5, tool0;
	MoveL Offs(p0,65.0,108.0, 0), v10, z5, tool0;
	MoveL Offs(p0,65.0,108.0, 0), v10, z5, tool0;
	MoveL Offs(p0,63.0,110.0, 0), v10, z5, tool0;
	MoveL Offs(p0,63.0,111.0, 0), v10, z5, tool0;
	MoveL Offs(p0,62.0,112.0, 0), v10, z5, tool0;
	MoveL Offs(p0,62.0,113.0, 0), v10, z5, tool0;
	MoveL Offs(p0,62.0,114.0, 0), v10, z5, tool0;
	MoveL Offs(p0,61.0,114.0, 0), v10, z5, tool0;
	MoveL Offs(p0,61.0,115.0, 0), v10, z5, tool0;
	MoveL Offs(p0,63.0,114.0, 0), v10, z5, tool0;
	MoveJ Offs(p0,63.0,114.0, 20), v10, z1, tool0;
	MoveJ Offs(p0,69.0,114.0, 20), v10, z1, tool0;
	MoveJ Offs(p0,69.0,114.0, 0), v10, z1, tool0;
	MoveL Offs(p0,72.0,113.0, 0), v10, z5, tool0;
	MoveL Offs(p0,70.0,111.0, 0), v10, z5, tool0;
	MoveL Offs(p0,67.0,110.0, 0), v10, z5, tool0;
	MoveL Offs(p0,67.0,110.0, 0), v10, z5, tool0;
	MoveL Offs(p0,67.0,110.0, 0), v10, z5, tool0;
	MoveL Offs(p0,66.0,110.0, 0), v10, z5, tool0;
	MoveL Offs(p0,66.0,111.0, 0), v10, z5, tool0;
	MoveL Offs(p0,65.0,111.0, 0), v10, z5, tool0;
	MoveL Offs(p0,65.0,112.0, 0), v10, z5, tool0;
	MoveL Offs(p0,64.0,114.0, 0), v10, z5, tool0;
	MoveL Offs(p0,64.0,114.0, 0), v10, z5, tool0;
	MoveL Offs(p0,64.0,114.0, 0), v10, z5, tool0;
	MoveL Offs(p0,64.0,115.0, 0), v10, z5, tool0;
	MoveL Offs(p0,65.0,115.0, 0), v10, z5, tool0;
	MoveL Offs(p0,65.0,115.0, 0), v10, z5, tool0;
	MoveL Offs(p0,67.0,114.0, 0), v10, z5, tool0;
	MoveL Offs(p0,68.0,114.0, 0), v10, z5, tool0;
	MoveL Offs(p0,68.0,114.0, 0), v10, z5, tool0;
	MoveL Offs(p0,69.0,114.0, 0), v10, z5, tool0;
	MoveL Offs(p0,69.0,114.0, 0), v10, z5, tool0;
	MoveJ Offs(p0,69.0,114.0, 20), v10, z1, tool0;
	MoveJ Offs(p0,29.0,114.0, 20), v10, z1, tool0;
	MoveJ Offs(p0,29.0,114.0, 0), v10, z1, tool0;
	MoveL Offs(p0,30.0,113.0, 0), v10, z5, tool0;
	MoveL Offs(p0,30.0,114.0, 0), v10, z5, tool0;
	MoveL Offs(p0,33.0,110.0, 0), v10, z5, tool0;
	MoveL Offs(p0,33.0,109.0, 0), v10, z5, tool0;
	MoveL Offs(p0,32.0,107.0, 0), v10, z5, tool0;
	MoveL Offs(p0,32.0,106.0, 0), v10, z5, tool0;
	MoveL Offs(p0,31.0,105.0, 0), v10, z5, tool0;
	MoveL Offs(p0,31.0,103.0, 0), v10, z5, tool0;
	MoveL Offs(p0,30.0,102.0, 0), v10, z5, tool0;
	MoveL Offs(p0,30.0,101.0, 0), v10, z5, tool0;
	MoveL Offs(p0,28.0,99.0, 0), v10, z5, tool0;
	MoveL Offs(p0,28.0,98.0, 0), v10, z5, tool0;
	MoveL Offs(p0,27.0,97.0, 0), v10, z5, tool0;
	MoveL Offs(p0,27.0,96.0, 0), v10, z5, tool0;
	MoveL Offs(p0,26.0,96.0, 0), v10, z5, tool0;
	MoveL Offs(p0,26.0,95.0, 0), v10, z5, tool0;
	MoveL Offs(p0,26.0,95.0, 0), v10, z5, tool0;
	MoveL Offs(p0,26.0,96.0, 0), v10, z5, tool0;
	MoveL Offs(p0,26.0,98.0, 0), v10, z5, tool0;
